(* Netzzustand Kaltwasser *)
IF Aktor_Netze_Anford.Kaltwasser.Aktiv THEN
	Zustand_Netz_KW.Temp_Max					:= MAX(Zustand_Netz_KW.Temp_Max, Aktor_Netze_Anford.Kaltwasser.Temp_Oben);
	Zustand_Netz_KW.Temp_Min					:= MIN(Zustand_Netz_KW.Temp_Min, Aktor_Netze_Anford.Kaltwasser.Temp_Unten);
	Zustand_Netz_KW.Regelung_Sollw_Oben_Max	:= MIN( Zustand_Netz_KW.Regelung_Sollw_Oben_Max, Aktor_Netze_Anford.Kaltwasser.Temp_Oben_Max);
	Zustand_Netz_KW.Regelung_Sollw_Oben_Min		:= MAX( Zustand_Netz_KW.Regelung_Sollw_Oben_Min, Aktor_Netze_Anford.Kaltwasser.Temp_Oben_Min);
	Zustand_Netz_KW.Regelung_Sollw_Unten_Max	:= MIN( Zustand_Netz_KW.Regelung_Sollw_Unten_Max, Aktor_Netze_Anford.Kaltwasser.Temp_Unten_Max);
	Zustand_Netz_KW.Regelung_Sollw_Unten_Min	:= MAX( Zustand_Netz_KW.Regelung_Sollw_Unten_Min, Aktor_Netze_Anford.Kaltwasser.Temp_Unten_Max);
END_IF
(* Netzzustand Warmwasser *)
IF Aktor_Netze_Anford.Warmwasser.Aktiv THEN
	Zustand_Netz_WW.Temp_Max					:= MAX(Zustand_Netz_WW.Temp_Max, Aktor_Netze_Anford.Kaltwasser.Temp_Oben);
	Zustand_Netz_WW.Temp_Min					:= MIN(Zustand_Netz_WW.Temp_Min, Aktor_Netze_Anford.Kaltwasser.Temp_Unten);
	Zustand_Netz_WW.Regelung_Sollw_Oben_Max	:= MIN( Zustand_Netz_WW.Regelung_Sollw_Oben_Max, Aktor_Netze_Anford.Kaltwasser.Temp_Oben_Max);
	Zustand_Netz_WW.Regelung_Sollw_Oben_Min	:= MAX( Zustand_Netz_WW.Regelung_Sollw_Oben_Min, Aktor_Netze_Anford.Kaltwasser.Temp_Oben_Min);
	Zustand_Netz_WW.Regelung_Sollw_Unten_Max	:= MIN( Zustand_Netz_WW.Regelung_Sollw_Unten_Max, Aktor_Netze_Anford.Kaltwasser.Temp_Unten_Max);
	Zustand_Netz_WW.Regelung_Sollw_Unten_Min	:= MAX( Zustand_Netz_WW.Regelung_Sollw_Unten_Min, Aktor_Netze_Anford.Kaltwasser.Temp_Unten_Max);
END_IF
(* Netzzustand Heisswasser *)
IF Aktor_Netze_Anford.Heisswasser.Aktiv THEN
	Zustand_Netz_HW.Temp_Max					:= MAX(Zustand_Netz_HW.Temp_Max, Aktor_Netze_Anford.Kaltwasser.Temp_Oben);
	Zustand_Netz_HW.Temp_Min					:= MIN(Zustand_Netz_HW.Temp_Min, Aktor_Netze_Anford.Kaltwasser.Temp_Unten);
	Zustand_Netz_HW.Regelung_Sollw_Oben_Max	:= MIN( Zustand_Netz_HW.Regelung_Sollw_Oben_Max, Aktor_Netze_Anford.Kaltwasser.Temp_Oben_Max);
	Zustand_Netz_HW.Regelung_Sollw_Oben_Min	:= MAX( Zustand_Netz_HW.Regelung_Sollw_Oben_Min, Aktor_Netze_Anford.Kaltwasser.Temp_Oben_Min);
	Zustand_Netz_HW.Regelung_Sollw_Unten_Max	:= MIN( Zustand_Netz_HW.Regelung_Sollw_Unten_Max, Aktor_Netze_Anford.Kaltwasser.Temp_Unten_Max);
	Zustand_Netz_HW.Regelung_Sollw_Unten_Min	:= MAX( Zustand_Netz_HW.Regelung_Sollw_Unten_Min, Aktor_Netze_Anford.Kaltwasser.Temp_Unten_Max);
END_IF;

Hysterese_Parameter.tTaskCycleTime	:= GA_global.Zeit_TaskCycle;
Hysterese_Parameter.tCtrlCycleTime		:= DINT_TO_TIME(Parameter.Kennlinie_Tctr);
Hysterese_Parameter.fHysteresisRange	:= 1;	(* 1 K *)

(* Initialisieren *)
Zustand.EIN_Anford		:= FALSE;
Zustand.EIN_Prioritaet		:= 0;
Zustand.AUS_Anford		:= FALSE;
Zustand.AUS_Prioritaet		:= 0;

(* Netzregelung Kaltwasser *)
IF( Parameter.Regelung_Netz_KW.Heizung AND Stellwert_Netz_KW.Leistung > 0 ) THEN
	Hysterese_Parameter.fHysteresisRange	:= Parameter.Regelung_Netz_KW.Hysterese_Heizung;
	Hysterese_KW_Heizung(
		fSetpointValue	:= Parameter.Regelung_Netz_KW.Grenzwert_Heizung,
		fActualValue		:= Stellwert_Netz_KW.Leistung,
		bSync			:= FALSE,
		eMode			:= eCTRL_MODE_ACTIVE,
		stParams		:= Hysterese_Parameter
	);
	IF( Hysterese_KW_Heizung.bOut ) THEN
		IF( Parameter.Regelung_Netz_KW.Invertiert_Heizung AND Parameter.Regelung_Netz_KW.Prioritaet_Heizung >= Zustand.AUS_Prioritaet) THEN
			Zustand.AUS_Anford		:= TRUE;
			Zustand.AUS_Prioritaet		:= Parameter.Regelung_Netz_KW.Prioritaet_Heizung;
		ELSIF( NOT Parameter.Regelung_Netz_KW.Invertiert_Heizung AND Parameter.Regelung_Netz_KW.Prioritaet_Heizung >= Zustand.EIN_Prioritaet) THEN
			Zustand.EIN_Anford		:= TRUE;
			Zustand.EIN_Prioritaet		:= Parameter.Regelung_Netz_KW.Prioritaet_Heizung;
		END_IF;
	END_IF;
ELSIF( Parameter.Regelung_Netz_KW.Heizung AND Stellwert_Netz_KW.Leistung < 0 ) THEN
	Hysterese_Parameter.fHysteresisRange	:= Parameter.Regelung_Netz_KW.Hysterese_Kuehlung;
	Hysterese_KW_Kuehlung(
		fSetpointValue	:= (-1) * Parameter.Regelung_Netz_KW.Grenzwert_Kuehlung,
		fActualValue		:= (-1) * Stellwert_Netz_KW.Leistung,
		bSync			:= FALSE,
		eMode			:= eCTRL_MODE_ACTIVE,
		stParams		:= Hysterese_Parameter
	);
	IF( Hysterese_KW_Kuehlung.bOut ) THEN
		IF( Parameter.Regelung_Netz_KW.Invertiert_Kuehlung AND Parameter.Regelung_Netz_KW.Prioritaet_Kuehlung >= Zustand.AUS_Prioritaet) THEN
			Zustand.AUS_Anford		:= TRUE;
			Zustand.AUS_Prioritaet		:= Parameter.Regelung_Netz_KW.Prioritaet_Kuehlung;
		ELSIF( NOT Parameter.Regelung_Netz_KW.Invertiert_Kuehlung AND Parameter.Regelung_Netz_KW.Prioritaet_Kuehlung >= Zustand.EIN_Prioritaet) THEN
			Zustand.EIN_Anford		:= TRUE;
			Zustand.EIN_Prioritaet		:= Parameter.Regelung_Netz_KW.Prioritaet_Kuehlung;
		END_IF;
	END_IF;
END_IF;

(* Netzregelung Warmwasser *)
IF( Parameter.Regelung_Netz_WW.Heizung AND Stellwert_Netz_WW.Leistung > 0 ) THEN
	Hysterese_Parameter.fHysteresisRange	:= Parameter.Regelung_Netz_WW.Hysterese_Heizung;
	Hysterese_WW_Heizung(
		fSetpointValue	:= Parameter.Regelung_Netz_WW.Grenzwert_Heizung,
		fActualValue		:= Stellwert_Netz_WW.Leistung,
		bSync			:= FALSE,
		eMode			:= eCTRL_MODE_ACTIVE,
		stParams		:= Hysterese_Parameter
	);
	IF( Hysterese_WW_Heizung.bOut ) THEN
		IF( Parameter.Regelung_Netz_WW.Invertiert_Heizung AND Parameter.Regelung_Netz_WW.Prioritaet_Heizung >= Zustand.AUS_Prioritaet) THEN
			Zustand.AUS_Anford		:= TRUE;
			Zustand.AUS_Prioritaet		:= Parameter.Regelung_Netz_WW.Prioritaet_Heizung;
		ELSIF( NOT Parameter.Regelung_Netz_WW.Invertiert_Heizung AND Parameter.Regelung_Netz_WW.Prioritaet_Heizung >= Zustand.EIN_Prioritaet) THEN
			Zustand.EIN_Anford		:= TRUE;
			Zustand.EIN_Prioritaet		:= Parameter.Regelung_Netz_WW.Prioritaet_Heizung;
		END_IF;
	END_IF;
ELSIF( Parameter.Regelung_Netz_WW.Heizung AND Stellwert_Netz_WW.Leistung < 0 ) THEN
	Hysterese_Parameter.fHysteresisRange	:= Parameter.Regelung_Netz_WW.Hysterese_Kuehlung;
	Hysterese_WW_Kuehlung(
		fSetpointValue	:= (-1) * Parameter.Regelung_Netz_WW.Grenzwert_Kuehlung,
		fActualValue		:= (-1) * Stellwert_Netz_WW.Leistung,
		bSync			:= FALSE,
		eMode			:= eCTRL_MODE_ACTIVE,
		stParams		:= Hysterese_Parameter
	);
	IF( Hysterese_WW_Kuehlung.bOut ) THEN
		IF( Parameter.Regelung_Netz_WW.Invertiert_Kuehlung AND Parameter.Regelung_Netz_WW.Prioritaet_Kuehlung >= Zustand.AUS_Prioritaet) THEN
			Zustand.AUS_Anford		:= TRUE;
			Zustand.AUS_Prioritaet		:= Parameter.Regelung_Netz_WW.Prioritaet_Kuehlung;
		ELSIF( NOT Parameter.Regelung_Netz_WW.Invertiert_Kuehlung AND Parameter.Regelung_Netz_WW.Prioritaet_Kuehlung >= Zustand.EIN_Prioritaet) THEN
			Zustand.EIN_Anford		:= TRUE;
			Zustand.EIN_Prioritaet		:= Parameter.Regelung_Netz_WW.Prioritaet_Kuehlung;
		END_IF;
	END_IF;
END_IF;

(* Netzregelung Heisswasser *)
IF( Parameter.Regelung_Netz_HW.Heizung AND Stellwert_Netz_HW.Leistung > 0 ) THEN
	Hysterese_Parameter.fHysteresisRange	:= Parameter.Regelung_Netz_HW.Hysterese_Heizung;
	Hysterese_HW_Heizung(
		fSetpointValue	:= Parameter.Regelung_Netz_HW.Grenzwert_Heizung,
		fActualValue		:= Stellwert_Netz_HW.Leistung,
		bSync			:= FALSE,
		eMode			:= eCTRL_MODE_ACTIVE,
		stParams		:= Hysterese_Parameter
	);
	IF( Hysterese_HW_Heizung.bOut ) THEN
		IF( Parameter.Regelung_Netz_HW.Invertiert_Heizung AND Parameter.Regelung_Netz_HW.Prioritaet_Heizung >= Zustand.AUS_Prioritaet) THEN
			Zustand.AUS_Anford		:= TRUE;
			Zustand.AUS_Prioritaet		:= Parameter.Regelung_Netz_HW.Prioritaet_Heizung;
		ELSIF( NOT Parameter.Regelung_Netz_HW.Invertiert_Heizung AND Parameter.Regelung_Netz_HW.Prioritaet_Heizung >= Zustand.EIN_Prioritaet) THEN
			Zustand.EIN_Anford		:= TRUE;
			Zustand.EIN_Prioritaet		:= Parameter.Regelung_Netz_HW.Prioritaet_Heizung;
		END_IF;
	END_IF;
ELSIF( Parameter.Regelung_Netz_HW.Heizung AND Stellwert_Netz_HW.Leistung < 0 ) THEN
	Hysterese_Parameter.fHysteresisRange	:= Parameter.Regelung_Netz_HW.Hysterese_Kuehlung;
	Hysterese_HW_Kuehlung(
		fSetpointValue	:= (-1) * Parameter.Regelung_Netz_HW.Grenzwert_Kuehlung,
		fActualValue		:= (-1) * Stellwert_Netz_HW.Leistung,
		bSync			:= FALSE,
		eMode			:= eCTRL_MODE_ACTIVE,
		stParams		:= Hysterese_Parameter
	);
	IF( Hysterese_HW_Kuehlung.bOut ) THEN
		IF( Parameter.Regelung_Netz_HW.Invertiert_Kuehlung AND Parameter.Regelung_Netz_HW.Prioritaet_Kuehlung >= Zustand.AUS_Prioritaet) THEN
			Zustand.AUS_Anford		:= TRUE;
			Zustand.AUS_Prioritaet		:= Parameter.Regelung_Netz_HW.Prioritaet_Kuehlung;
		ELSIF( NOT Parameter.Regelung_Netz_HW.Invertiert_Kuehlung AND Parameter.Regelung_Netz_HW.Prioritaet_Kuehlung >= Zustand.EIN_Prioritaet) THEN
			Zustand.EIN_Anford		:= TRUE;
			Zustand.EIN_Prioritaet		:= Parameter.Regelung_Netz_HW.Prioritaet_Kuehlung;
		END_IF;
	END_IF;
END_IF;



(* Stellwert bestimmen *)
Stellwert.Betrieb	:= Zustand.EIN_Anford AND NOT (Zustand.AUS_Anford AND (Zustand.AUS_Prioritaet > Zustand.EIN_Prioritaet));

END_FUNCTION_BLOCK

// ---- POUs/Management/FB_MGMT_Logik.TcPOU


FUNCTION_BLOCK FB_MGMT_Logik
VAR_IN_OUT
	Steuerung	: ST_FB_MGMT_Steuerung;
	Zustand		: ST_FB_MGMT_Zustand;
END_VAR
VAR_INPUT
	Parameter	: ST_FB_MGMT_Parameter;
END_VAR
VAR_OUTPUT
END_VAR
VAR
END_VAR

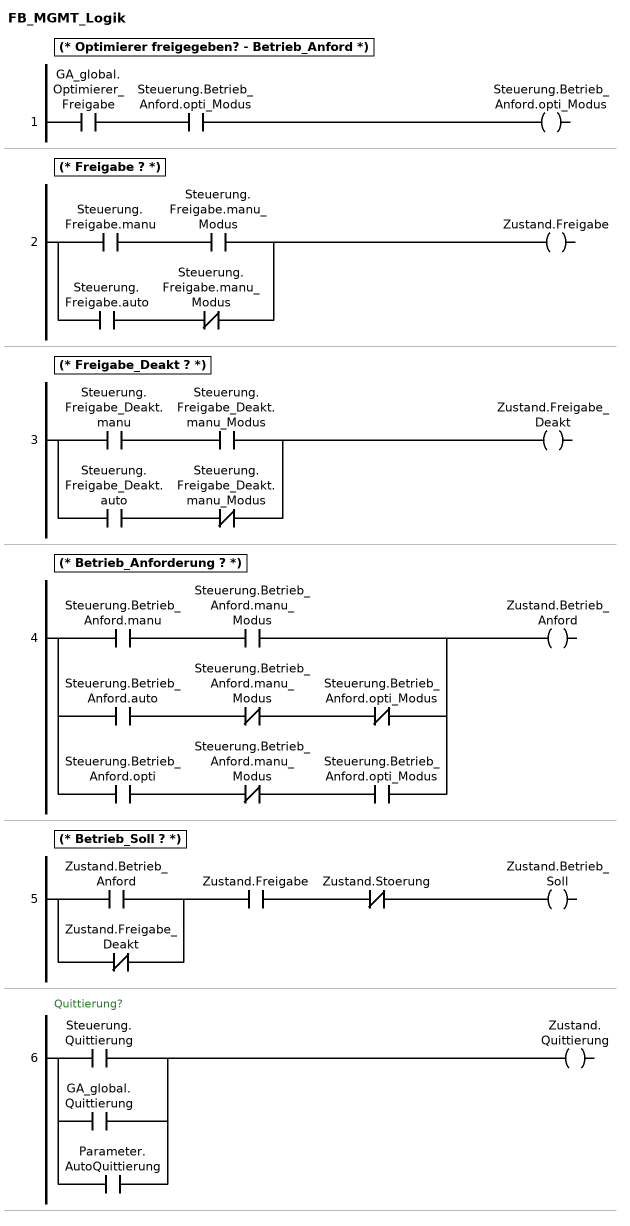
// NETWORK 1
// label: (* Optimierer freigegeben? - Betrieb_Anford *)
Steuerung.Betrieb_Anford.opti_Modus := GA_global.Optimierer_Freigabe AND Steuerung.Betrieb_Anford.opti_Modus;

// NETWORK 2
// label: (* Freigabe ? *)
Zustand.Freigabe := Steuerung.Freigabe.manu AND Steuerung.Freigabe.manu_Modus OR Steuerung.Freigabe.auto AND NOT Steuerung.Freigabe.manu_Modus;

// NETWORK 3
// label: (* Freigabe_Deakt ? *)
Zustand.Freigabe_Deakt := Steuerung.Freigabe_Deakt.manu AND Steuerung.Freigabe_Deakt.manu_Modus OR Steuerung.Freigabe_Deakt.auto AND NOT Steuerung.Freigabe_Deakt.manu_Modus;

// NETWORK 4
// label: (* Betrieb_Anforderung ? *)
Zustand.Betrieb_Anford := Steuerung.Betrieb_Anford.manu AND Steuerung.Betrieb_Anford.manu_Modus OR Steuerung.Betrieb_Anford.auto AND NOT Steuerung.Betrieb_Anford.manu_Modus AND NOT Steuerung.Betrieb_Anford.opti_Modus OR Steuerung.Betrieb_Anford.opti AND NOT Steuerung.Betrieb_Anford.manu_Modus AND Steuerung.Betrieb_Anford.opti_Modus;

// NETWORK 5
// label: (* Betrieb_Soll ? *)
Zustand.Betrieb_Soll := (Zustand.Betrieb_Anford OR NOT Zustand.Freigabe_Deakt) AND Zustand.Freigabe AND NOT Zustand.Stoerung;

// NETWORK 6
// Quittierung?
Zustand.Quittierung := Steuerung.Quittierung OR GA_global.Quittierung OR Parameter.AutoQuittierung;

END_FUNCTION_BLOCK

// ---- POUs/Management/FB_MGMT_Ablaufsteuerung.TcPOU
FUNCTION_BLOCK FB_MGMT_Ablaufsteuerung
VAR_IN_OUT
	Zustand				: ST_FB_MGMT_Zustand;
	Stellwert			: ST_FB_MGMT_Stellwert;
	Steuerung			: ST_FB_MGMT_Steuerung;
END_VAR
VAR_INPUT
END_VAR
VAR_OUTPUT
END_VAR
VAR
END_VAR

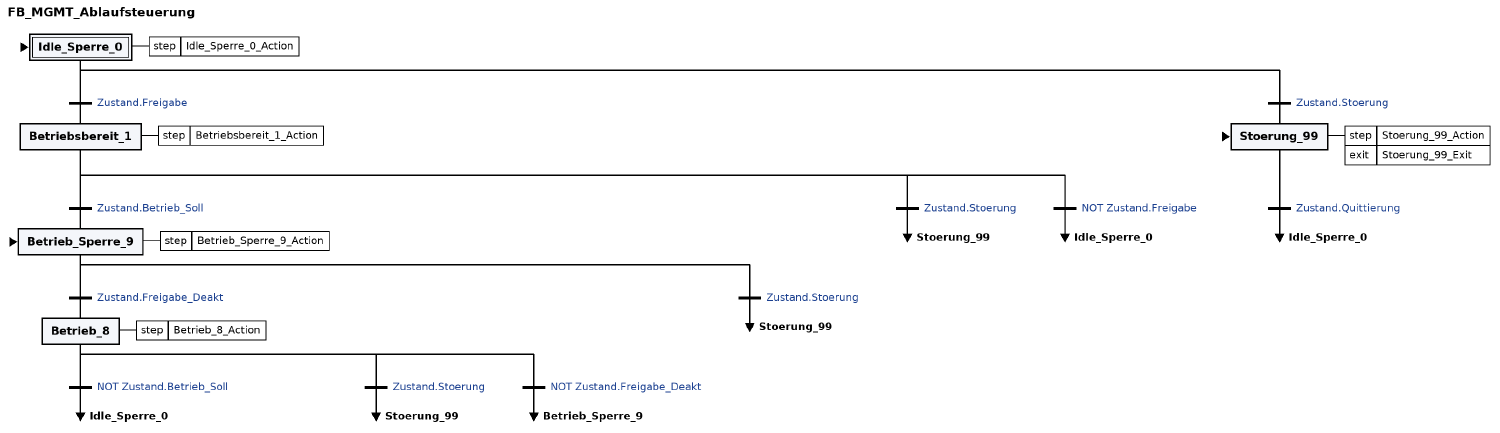
INITIAL_STEP Idle_Sperre_0:
    Idle_Sperre_0_Action(N);  // step action
END_STEP
TRANSITION FROM Idle_Sperre_0 TO Betriebsbereit_1
    := Zustand.Freigabe;
END_TRANSITION
TRANSITION FROM Idle_Sperre_0 TO Stoerung_99
    := Zustand.Stoerung;
END_TRANSITION
STEP Stoerung_99:
    Stoerung_99_Action(N);  // step action
    Stoerung_99_Exit(P0);  // exit action
END_STEP
TRANSITION FROM Stoerung_99 TO Idle_Sperre_0
    := Zustand.Quittierung;
END_TRANSITION
STEP Betriebsbereit_1:
    Betriebsbereit_1_Action(N);  // step action
END_STEP
TRANSITION FROM Betriebsbereit_1 TO Betrieb_Sperre_9
    := Zustand.Betrieb_Soll;
END_TRANSITION
TRANSITION FROM Betriebsbereit_1 TO Stoerung_99
    := Zustand.Stoerung;
END_TRANSITION
TRANSITION FROM Betriebsbereit_1 TO Idle_Sperre_0
    := NOT Zustand.Freigabe;
END_TRANSITION
STEP Betrieb_Sperre_9:
    Betrieb_Sperre_9_Action(N);  // step action
END_STEP
TRANSITION FROM Betrieb_Sperre_9 TO Betrieb_8
    := Zustand.Freigabe_Deakt;
END_TRANSITION
TRANSITION FROM Betrieb_Sperre_9 TO Stoerung_99
    := Zustand.Stoerung;
END_TRANSITION
STEP Betrieb_8:
    Betrieb_8_Action(N);  // step action
END_STEP
TRANSITION FROM Betrieb_8 TO Idle_Sperre_0
    := NOT Zustand.Betrieb_Soll;
END_TRANSITION
TRANSITION FROM Betrieb_8 TO Stoerung_99
    := Zustand.Stoerung;
END_TRANSITION
TRANSITION FROM Betrieb_8 TO Betrieb_Sperre_9
    := NOT Zustand.Freigabe_Deakt;
END_TRANSITION

ACTION Betrieb_8_Action:
(* Stellwert setzen *)
Stellwert.Betrieb				:= TRUE;
Zustand.Betrieb				:= TRUE;

(* Zustand setzen *)
Zustand.Status				:= E_MGMT_Zustand_Status_Betrieb;
END_ACTION

ACTION Betrieb_Sperre_9_Action:
(* Stellwert setzen *)
Stellwert.Betrieb				:= TRUE;
Zustand.Betrieb				:= TRUE;

(* Zustand setzen *)
Zustand.Status				:= E_MGMT_Zustand_Status_Betrieb_Sperre;
END_ACTION

ACTION Betriebsbereit_1_Action:
(* Stellwert setzen *)
Stellwert.Betrieb		:= FALSE;
Zustand.Betrieb		:= FALSE;

(* Zustand setzen *)
Zustand.Status			:= E_MGMT_Zustand_Status_Betriebsbereit;
END_ACTION

ACTION Idle_Sperre_0_Action:
(* Stellwert setzen *)
Stellwert.Betrieb		:= FALSE;
Zustand.Betrieb			:= FALSE;

(* Zustand setzen *)
Zustand.Status				:= E_MGMT_Zustand_Status_Idle_Sperre;

(* Quittierungszustand auf False setzen, damit das System bei einer erneuten Störung nicht direkt wieder angeschaltet wird *)
Steuerung.Quittierung	:= FALSE;
END_ACTION

ACTION Stoerung_99_Action:
(* Stellwert setzen *)
Stellwert.Betrieb			:= FALSE;
Zustand.Betrieb			:= FALSE;

(* Zustand setzen *)
Zustand.Stoerung			:= TRUE;
Zustand.Status			:= E_MGMT_Zustand_Status_Stoerung;
END_ACTION

ACTION Stoerung_99_Exit:
Zustand.Stoerung	:= FALSE;
END_ACTION

END_FUNCTION_BLOCK

// ---- POUs/Management/FB_MGMT_Sollwertscheck.TcPOU
FUNCTION_BLOCK FB_MGMT_Sollwertscheck
VAR_IN_OUT
	Zustand		: ST_FB_MGMT_Zustand;
END_VAR
VAR_INPUT
	Steuerung	: ST_FB_MGMT_Steuerung;
	Parameter	: ST_FB_MGMT_Parameter;
END_VAR
VAR

END_VAR

(* Priorisierung Regelung_Modus *)
IF(Steuerung.Regelung_Modus.manu_Modus) THEN
	Zustand.Regelung_Modus := Steuerung.Regelung_Modus.manu;
ELSIF(Steuerung.Regelung_Modus.opti_Modus) THEN
	Zustand.Regelung_Modus := Steuerung.Regelung_Modus.opti;
ELSE
	Zustand.Regelung_Modus := Steuerung.Regelung_Modus.auto;
END_IF;
(* Priorisierung Regelung_Sollwert *)
IF(Steuerung.Regelung_Sollw.manu_Modus) THEN
	Zustand.Regelung_Sollw_Anford := Steuerung.Regelung_Sollw.manu;
ELSIF(Steuerung.Regelung_Sollw.opti_Modus) THEN
	Zustand.Regelung_Sollw_Anford := Steuerung.Regelung_Sollw.opti;
ELSE
	Zustand.Regelung_Sollw_Anford := Steuerung.Regelung_Sollw.auto;
END_IF;

(*Berechnung Sollwert mithilfe von Netze*)

(*Heizen*)

Zustand.Regelung_Sollw_BHKW_WBZ := Zustand.Heisswasser_3xx_Zustand_Regelung_Sollw;
Zustand.Regelung_Sollw_BHKW_MBZ := Zustand.Heisswasser_3xx_Zustand_Regelung_Sollw - 2;
Zustand.Regelung_Sollw_BWT:= Zustand.Heisswasser_3xx_Zustand_Regelung_Sollw - 4;

(*Warmnetz*)
Zustand.Regelung_Sollw_PTW1:= Zustand.Warmwasser_2xx_Zustand_Regelung_Sollw;
Zustand.Regelung_Sollw_WP_gruennetz :=  Zustand.Warmwasser_2xx_Zustand_Regelung_Sollw - 3;
Zustand.Regelung_Sollw_gruennetz_Kuehlung:=Zustand.Warmwasser_2xx_Zustand_Regelung_Sollw_Max;


(*Kühlen*)
Zustand.Regelung_Sollw_blaunetz_Kuehlung:= Zustand.Kaltwasser_1xx_Zustand_Regelung_Sollw;
Zustand.Regelung_Sollw_Kuehlung_KKKW := MIN(Zustand.Kaltwasser_1xx_Zustand_Regelung_Sollw + 3, Zustand.Temp_KRITIKAL_OBEN_TEMP_Kaltnetz)  ;
Zustand.Regelung_Sollw_WP_945 := MAX(Zustand.Kaltwasser_1xx_Zustand_Regelung_Sollw, Zustand.Temp_KRITIKAL_UNTEN_TEMP_Kaltnetz );

END_FUNCTION_BLOCK

// ---- POUs/Management/FB_MGMT_Regelung.TcPOU
FUNCTION_BLOCK FB_MGMT_Regelung
VAR_IN_OUT
	Stellwert	: ST_FB_MGMT_Stellwert;
	Zustand		: ST_FB_MGMT_Zustand;
END_VAR
VAR_INPUT
	Steuerung	: ST_FB_MGMT_Steuerung;
	Parameter	: ST_FB_MGMT_Parameter;
END_VAR
VAR_OUTPUT
END_VAR
VAR
(*Hysterese Heizung*)
	Hysterese_BHKW_MBZ 					: FB_CTRL_2POINT; (*BHKW mit mehrerer Betriebzeit*)
	Hysterese_Parameter_BHKW_MBZ		: ST_CTRL_2POINT_PARAMS; (*BHKW mit mehrerer Betriebzeit*)
	Hysterese_BHKW_WBZ 					: FB_CTRL_2POINT; (*BHKW mit wenigerer Betriebzeit*)
	Hysterese_Parameter_BHKW_WBZ 		: ST_CTRL_2POINT_PARAMS; (*BHKW mit wenigerer Betriebzeit*)
	Hysterese_PWT_915 					: FB_CTRL_2POINT;
	Hysterese_Parameter_PWT_915 		: ST_CTRL_2POINT_PARAMS;
	Hysterese_BWT 						: FB_CTRL_2POINT;
	Hysterese_Parameter_BWT		 		: ST_CTRL_2POINT_PARAMS;
	Hysterese_WP_gruennetz				: FB_CTRL_2POINT;
	Hysterese_Parameter_WP_gruennetz	: ST_CTRL_2POINT_PARAMS;

(*Hysterese Kuehlung*)
	Hysterese_Kuehlung_KKKW                 : FB_CTRL_2POINT;
    Hysterese_Parameter_Kuehlung_KKKW       : ST_CTRL_2POINT_PARAMS;
	Hysterese_WP_945						: FB_CTRL_2POINT;
	Hysterese_Parameter_WP_945				: ST_CTRL_2POINT_PARAMS;

	WaermePumpe_Anforderung_gruennetz: BOOL;
	WaermePumpe_Anforderung_blaunetz: BOOL;

	Hysterese_BHKW_921: BOOL;
	t: REAL;
	Wechsel_Erlaubnis: BOOL; (*wenn Wechsel_Erlaubnis==true ist, dann darf Wechsel zwischen Hysterese erfolgen. Wechsel_Erlaubnis wird erst nach 24 Stunden nach dem letzten Wechsel True*)
	tstunde: REAL; (*Wenn die Hysterese für BHKW gewechselt werden*)
	ttag: REAL; (*Wenn die Hysterese für BHKW gewechselt werden*)
    aktuell_Modus: INT; (*Wenn diese Variable 1 ist, dann Output.BHKW2=MBZ und wenn 2 ist, dann Output.BHKW1=WBZ*)

    Kuehlung_Erlaubnis_KKKW    : BOOL; (*Wenn die Isttemperatur vom blauen Netz ist mehr als 3 Grad mehr als Solltemperatur, dann Chiller wird abgeschaltet. *)
END_VAR

(*Hysterese_Regelung für BHKW_MBZ(BHKW mit mehrerer Betriebzeit), Hysterese von Zustand.Regelung_Sollw_BHKW_MBZ-Range/2 bis Zustand.Regelung_Sollw_BHKW_MBZ+Range/2 °C*)

Hysterese_Parameter_BHKW_MBZ.fHysteresisRange := Parameter.Hysterese_BHKW_Range;
Hysterese_Parameter_BHKW_MBZ.tTaskCycleTime	:= GA_global.Zeit_TaskCycle; (* Zykluszeit FB = globaler Zykluszeit*)
Hysterese_Parameter_BHKW_MBZ.tCtrlCycleTime := GA_global.Zeit_TaskCycle;

Hysterese_BHKW_MBZ(
	fSetpointValue  := Zustand.Regelung_Sollw_BHKW_MBZ,
	fActualValue    := Zustand.Temp_Hysterese_BHKW_A,
	eMode			:= eCTRL_MODE_ACTIVE,
	stParams		:= Hysterese_Parameter_BHKW_MBZ
);

(*Beim Aufheizen wird auf untere Temperatur geregelt, beim Abkühlen wird auf obere Temperatur geregelt.*)

IF (Hysterese_BHKW_MBZ.bOut) THEN
Zustand.Temp_Hysterese_BHKW_A := Zustand.Temp_Unten_Heissnetz;
ELSE
Zustand.Temp_Hysterese_BHKW_A := Zustand.Temp_Oben_Heissnetz;
END_IF

(*Hysterese_Regelung für BHKW_WBZ(BHKW mit wenigerer Betriebzeit), Hysterese von Zustand.Regelung_Sollw_BHKW_WBZ-Range/2 bis Zustand.Regelung_Sollw_BHKW_WBZ+Range/2 °C*)

Hysterese_Parameter_BHKW_WBZ.fHysteresisRange := Parameter.Hysterese_BHKW_Range;
Hysterese_Parameter_BHKW_WBZ.tTaskCycleTime	:= GA_global.Zeit_TaskCycle; (* Zykluszeit FB = globaler Zykluszeit*)
Hysterese_Parameter_BHKW_WBZ.tCtrlCycleTime := GA_global.Zeit_TaskCycle;

Hysterese_BHKW_WBZ(
	fSetpointValue  := Zustand.Regelung_Sollw_BHKW_WBZ,
	fActualValue    := Zustand.Temp_Hysterese_BHKW_B,
	eMode			:= eCTRL_MODE_ACTIVE,
	stParams		:= Hysterese_Parameter_BHKW_WBZ
);

(*Beim Aufheizen wird auf untere Temperatur geregelt, beim Abkühlen wird auf obere Temperatur geregelt.*)

IF (Hysterese_BHKW_WBZ.bOut) THEN
Zustand.Temp_Hysterese_BHKW_B := Zustand.Temp_Unten_Heissnetz;
ELSE
Zustand.Temp_Hysterese_BHKW_B := Zustand.Temp_Oben_Heissnetz;
END_IF


(*BHKW mit wenigerer Betriebzeit übernimmt die höhere Hysterese*)

IF	(Wandler.System_Blockheizkraftwerk_922.BHKW_922.Zustand.Zeit_Betrieb>Wandler.System_Blockheizkraftwerk_921.BHKW_921.Zustand.Zeit_Betrieb) AND (Wechsel_Erlaubnis) THEN

Wechsel_Erlaubnis:=FALSE;
ttag:=GA_global.Systemzeit_Tag;
tstunde:=GA_global.Systemzeit_Stunde;
aktuell_Modus:=1;

ELSIF (Wandler.System_Blockheizkraftwerk_922.BHKW_922.Zustand.Zeit_Betrieb<Wandler.System_Blockheizkraftwerk_921.BHKW_921.Zustand.Zeit_Betrieb) AND (Wechsel_Erlaubnis) THEN

Wechsel_Erlaubnis:=FALSE;
ttag:=GA_global.Systemzeit_Tag;
tstunde:=GA_global.Systemzeit_Stunde;
aktuell_Modus:=2;

END_IF

CASE aktuell_Modus OF
1:
Stellwert.BHKW1_Anforderung := Hysterese_BHKW_WBZ.bOut;
Stellwert.BHKW2_Anforderung := Hysterese_BHKW_MBZ.bOut;

2:
Stellwert.BHKW1_Anforderung := Hysterese_BHKW_MBZ.bOut;
Stellwert.BHKW2_Anforderung := Hysterese_BHKW_WBZ.bOut;
END_CASE;

(*Wenn ein BHKW in Störung ist, dann übernimmt die andere seine Hysterese*)
IF (Zustand.BHKW921_Stoerung) AND (Stellwert.BHKW1_Anforderung) THEN
Stellwert.BHKW2_Anforderung := Stellwert.BHKW1_Anforderung;
ELSIF (Zustand.BHKW922_Stoerung) AND (Stellwert.BHKW2_Anforderung) THEN
Stellwert.BHKW1_Anforderung := Stellwert.BHKW2_Anforderung;
END_IF

(*Der Wechsel zwischen Hysterese darf nur einmal in 24 Stunden passieren.*)
t:= (GA_global.Systemzeit_Tag-ttag)*24 + GA_global.Systemzeit_Stunde-tstunde;

IF(t>24) THEN
Wechsel_Erlaubnis:=TRUE;
ELSE
Wechsel_Erlaubnis:= FALSE;
END_IF


(*Brennwerttherme an, Hysterese von Zustand.Regelung_Sollw_BWT-Range/2 bis Zustand.Regelung_Sollw_BWT+Range/2 °C*)
Hysterese_Parameter_BWT.fHysteresisRange := Parameter.Hysterese_BWT_Range;
Hysterese_Parameter_BWT.tTaskCycleTime	:= GA_global.Zeit_TaskCycle; (* Zykluszeit FB = globaler Zykluszeit*)
Hysterese_Parameter_BWT.tCtrlCycleTime := GA_global.Zeit_TaskCycle;

Hysterese_BWT(
	fSetpointValue  := Zustand.Regelung_Sollw_BWT,
	fActualValue    := Zustand.Temp_Hysterese_BWT,
	bSync			:= FALSE,
	eMode			:= eCTRL_MODE_ACTIVE,
	stParams		:= Hysterese_Parameter_BWT
);

Stellwert.BWT_Anforderung  := Hysterese_BWT.bOut;

(*Beim Aufheizen wird auf untere Temperatur geregelt, beim Abkühlen wird auf obere Temperatur geregelt.*)

IF (Hysterese_BWT.bOut) THEN
Zustand.Temp_Hysterese_BWT := Zustand.Temp_Unten_Heissnetz;
ELSE
Zustand.Temp_Hysterese_BWT := Zustand.Temp_Oben_Heissnetz;
END_IF


(*Wärmetauscher an, Hysterese von  Zustand.Regelung_Sollw_PTW1-Range/2 bis  Zustand.Regelung_Sollw_PTW1+Range/2 °C*)

Hysterese_Parameter_PWT_915.fHysteresisRange := Parameter.Hysterese_PTW1_Range;
Hysterese_Parameter_PWT_915.tTaskCycleTime	:= GA_global.Zeit_TaskCycle; (* Zykluszeit FB = globaler Zykluszeit*)
Hysterese_Parameter_PWT_915.tCtrlCycleTime := GA_global.Zeit_TaskCycle;

Hysterese_PWT_915(
	fSetpointValue  := Zustand.Regelung_Sollw_PTW1,
	fActualValue    := Zustand.Temp_Unten_Warmnetz,
	bSync			:= FALSE,
	eMode			:= eCTRL_MODE_ACTIVE,
	stParams		:= Hysterese_Parameter_PWT_915
);

Stellwert.PWT1_Anforderung  := Hysterese_PWT_915.bOut;

(*Wärmepumpe kannzum Kühlen des blauen Netzes oder zum Aufwärmen des gelben Netzes benutzt werden*)
(*Wärmepumpe an, Hysterese Regelung von Zustand.Regelung_Sollw_WP_gruennetz-Range/2 bis Zustand.Regelung_Sollw_WP_gruennetz+Range/2 °C*)



Hysterese_Parameter_WP_gruennetz.fHysteresisRange := Parameter.Hysterese_WP_gruennetz_Range;
Hysterese_Parameter_WP_gruennetz.tTaskCycleTime	:= GA_global.Zeit_TaskCycle; (* Zykluszeit FB = globaler Zykluszeit*)
Hysterese_Parameter_WP_gruennetz.tCtrlCycleTime := GA_global.Zeit_TaskCycle;

Hysterese_WP_gruennetz(
	fSetpointValue  := Zustand.Regelung_Sollw_WP_gruennetz,
	fActualValue    := Zustand.Temp_Unten_Warmnetz,
	bSync			:= FALSE,
	eMode			:= eCTRL_MODE_ACTIVE,
	stParams		:= Hysterese_Parameter_WP_gruennetz
);

(*Wenn die Temperatur des Balunetzes weniger als Kritikal_Unten_Temp ist, dann müssen Wärmepumpe ausgeschaltet werden*)
WaermePumpe_Anforderung_gruennetz  := Hysterese_WP_gruennetz.bOut AND (Zustand.Temp_Unten_Kaltnetz>Zustand.Temp_KRITIKAL_UNTEN_TEMP_Kaltnetz);


(*Hysterese_Regelung für Wärmepumpe blaunetz_Kuehlung*)
Hysterese_Parameter_WP_945.fHysteresisRange := Parameter.Hysterese_WP_Range;
Hysterese_Parameter_WP_945.tTaskCycleTime	:= GA_global.Zeit_TaskCycle;	(* Zykluszeit FB = globaler Zykluszeit*)
Hysterese_Parameter_WP_945.tCtrlCycleTime	:= GA_global.Zeit_TaskCycle;

Hysterese_WP_945(
	fSetpointValue 	:= Zustand.Regelung_Sollw_WP_945 - 1,
	fActualValue    := Zustand.Temp_Oben_Kaltnetz,
	bSync			:= FALSE,
	eMode			:= eCTRL_MODE_ACTIVE,
	stParams 		:= Hysterese_Parameter_WP_945
);

(*Wenn die Temperatur des Gruennetzes mehr als Kritikal_Oben_Temp ist, dann müssen Wärmepumpe ausgeschaltet werden*)
WaermePumpe_Anforderung_blaunetz := NOT Hysterese_WP_945.bOut AND NOT Hysterese_WP_945.bError AND (Zustand.Temp_Oben_Warmnetz<Zustand.Temp_KRITIKAL_OBEN_TEMP_Warmnetz) ;

Stellwert.Waermepumpe_945_Anforderung :=  WaermePumpe_Anforderung_gruennetz OR WaermePumpe_Anforderung_blaunetz;

(*Hysterese_Regelung für Kältekompressor Kaltwasser*)

Hysterese_Parameter_Kuehlung_KKKW.fHysteresisRange :=Parameter.Hysterese_KKKW_Kuehlung_Range;
Hysterese_Parameter_Kuehlung_KKKW.tTaskCycleTime	:= GA_global.Zeit_TaskCycle; (* Zykluszeit FB = globaler Zykluszeit*)
Hysterese_Parameter_Kuehlung_KKKW.tCtrlCycleTime := GA_global.Zeit_TaskCycle;

Hysterese_Kuehlung_KKKW(
	fSetpointValue  := Zustand.Regelung_Sollw_Kuehlung_KKKW,
	fActualValue    := Zustand.Temp_Oben_Kaltnetz,
	bSync			:= FALSE,
	eMode			:= eCTRL_MODE_ACTIVE,
	stParams		:= Hysterese_Parameter_Kuehlung_KKKW
);

(*Wenn die Kühlleistung vom Speicher nicht reicht, dann schaltet der Chiller an*)

IF (Zustand.Temp_Oben_Kaltnetz-Zustand.Regelung_Sollw_blaunetz_Kuehlung>3) THEN
Kuehlung_Erlaubnis_KKKW := TRUE;
ELSE
Kuehlung_Erlaubnis_KKKW := FALSE;
END_IF

Stellwert.Kuehlung_KKKW_Anforderung := NOT Hysterese_Kuehlung_KKKW.bOut AND NOT Hysterese_Kuehlung_KKKW.bError AND Kuehlung_Erlaubnis_KKKW ;


(*Entziehen der Freigabe, wenn Kritikal ObenTemperatur überschritten wird*)
(*
IF (Zustand.Temp_Oben_Heissnetz>Zustand.Temp_KRITIKAL_OBEN_TEMP_Heissnetz) THEN

Stellwert.BHKW1_Freigabe_Entziehung := TRUE;
Stellwert.BHKW2_Freigabe_Entziehung := TRUE;
Stellwert.BWT_Freigabe_Entziehung := TRUE;
GA_global.Optimierer_Freigabe := FALSE;
ELSE
Stellwert.BHKW1_Freigabe_Entziehung := FALSE;
Stellwert.BHKW2_Freigabe_Entziehung := FALSE;
Stellwert.BWT_Freigabe_Entziehung := FALSE;
(*GA_global.Optimierer_Freigabe := TRUE;*)
END_IF

IF (Zustand.Temp_Oben_Warmnetz>Zustand.Temp_KRITIKAL_OBEN_TEMP_Warmnetz) THEN

Stellwert.PWT1_Freigabe_Entziehung := TRUE;
Stellwert.WP_Freigabe_Entziehung := TRUE;
GA_global.Optimierer_Freigabe := FALSE;

ELSE
Stellwert.PWT1_Freigabe_Entziehung := FALSE;
Stellwert.WP_Freigabe_Entziehung := FALSE;

END_IF

IF Zustand.Temp_Unten_Kaltnetz<Zustand.Temp_KRITIKAL_UNTEN_TEMP_Kaltnetz THEN
GA_global.Optimierer_Freigabe := FALSE;
END_IF
*)

END_FUNCTION_BLOCK

// ---- POUs/Management/FB_Zuweisungen.TcPOU
FUNCTION_BLOCK FB_Zuweisungen
VAR_INPUT
END_VAR
VAR_IN_OUT
	Zustand		: ST_FB_MGMT_Zustand;
END_VAR
VAR_OUTPUT
END_VAR
VAR
END_VAR

Zustand.Temp_Speicher795:= Speicher.System_Betonspeicher_Kaltwasser_795.Betonspeicher_795.Zustand.Temp_oben;
Zustand.Temp_Oben_Heissnetz :=Netze.Heisswasser_3xx.Zustand.Temp_Oben;
Zustand.Temp_Unten_Heissnetz:= Netze.Heisswasser_3xx.Zustand.Temp_Unten;
Zustand.Temp_Oben_Warmnetz:= Netze.Warmwasser_2xx.Zustand.Temp_Oben;
Zustand.Temp_Unten_Warmnetz:=Netze.Warmwasser_2xx.Zustand.Temp_Unten;
Zustand.Temp_Oben_Kaltnetz:=Netze.Kaltwasser_1xx.Zustand.Temp_Oben;
Zustand.Temp_Unten_Kaltnetz:=Netze.Kaltwasser_1xx.Zustand.Temp_Unten;
Zustand.BHKW921_Stoerung:=Wandler.System_Blockheizkraftwerk_921.Zustand.Stoerung;
Zustand.BHKW922_Stoerung:=Wandler.System_Blockheizkraftwerk_922.Zustand.Stoerung;
Zustand.Temp_KRITIKAL_OBEN_TEMP_Heissnetz:=Netze.Heisswasser_3xx.Parameter.Regelung_Sollw_KRITIKAL_OBEN_TEMP;
Zustand.Temp_KRITIKAL_OBEN_TEMP_Warmnetz:= Netze.Warmwasser_2xx.Parameter.Regelung_Sollw_KRITIKAL_OBEN_TEMP;
Zustand.Temp_KRITIKAL_OBEN_TEMP_Kaltnetz:=Netze.Kaltwasser_1xx.Parameter.Regelung_Sollw_KRITIKAL_OBEN_TEMP;
Zustand.Temp_KRITIKAL_UNTEN_TEMP_Heissnetz:=Netze.Heisswasser_3xx.Parameter.Regelung_Sollw_KRITIKAL_UNTEN_TEMP;
Zustand.Temp_KRITIKAL_UNTEN_TEMP_Warmnetz:= Netze.Warmwasser_2xx.Parameter.Regelung_Sollw_KRITIKAL_UNTEN_TEMP;
Zustand.Temp_KRITIKAL_UNTEN_TEMP_Kaltnetz:=Netze.Kaltwasser_1xx.Parameter.Regelung_Sollw_KRITIKAL_UNTEN_TEMP;

Zustand.Heisswasser_3xx_Zustand_Regelung_Sollw:= Netze.Heisswasser_3xx.Zustand.Regelung_Sollw;
Zustand.Warmwasser_2xx_Zustand_Regelung_Sollw:=Netze.Warmwasser_2xx.Zustand.Regelung_Sollw;
Zustand.Warmwasser_2xx_Zustand_Regelung_Sollw_Max := Netze.Warmwasser_2xx.Zustand.Regelung_Sollw_Max;
Zustand.Kaltwasser_1xx_Zustand_Regelung_Sollw:=Netze.Kaltwasser_1xx.Zustand.Regelung_Sollw;

END_FUNCTION_BLOCK

// ---- POUs/FB_Initialisierungsroutine.TcPOU
FUNCTION_BLOCK FB_Initialisierungsroutine
VAR_OUTPUT
END_VAR
VAR

END_VAR

(*Management Parameter*)

Initialisierung.MGMT_Parameter.Temp_Max :=100; (*Grad Celsius*)
Initialisierung.MGMT_Parameter.Temp_Min :=0; (*Grad Celsius*)
Initialisierung.MGMT_Parameter.AutoQuittierung := 0;

(*Management Parameter- Heizen*)

Initialisierung.MGMT_Parameter.Hysterese_BHKW_Range := 3; (*Grad Celsius*) (*Range von die Hysterese für BHKW*)
Initialisierung.MGMT_Parameter.Hysterese_BWT_Range := 5; (*Grad Celsius*) (*Range von die Hysterese für BWT*)
Initialisierung.MGMT_Parameter.Hysterese_PTW1_Range := 3; (*Grad Celsius*) (*Range von die Hysterese für PWT*)


(*Management Parameter- Kühlen*)
Initialisierung.MGMT_Parameter.Hysterese_blaunetz_Kuehlung_Range := 2; (*Grad Celsius*) (*Range von Blaunetz_Hysterese *)
Initialisierung.MGMT_Parameter.Hysterese_KKKW_Kuehlung_Range := 2; (*Grad Celsius*) (*Range von Kältekompressor_Hysterese*)
Initialisierung.MGMT_Parameter.Hysterese_gruennetz_Kuehlung_Range := 2; (*Grad Celsius*) (*Range von Grünnetz_Hysterese*)
Initialisierung.MGMT_Parameter.Hysterese_WP_gruennetz_Range := 2; (*Grad Celsius*) (*Range von Wärmepumpe für gruenNetz *)
Initialisierung.MGMT_Parameter.Hysterese_WP_Range := 2; (*Grad Celsius*) (*Range von Hysterese_Regelung für Wärmepumpe blau_kuehlmodus_Kuehlung*)

(*Netze Parameter*)
Initialisierung.Netze_Parameter.Heisswasser.Regelung_Sollw_Max_Min := 50; (*Grad Celsius*)
Initialisierung.Netze_Parameter.Heisswasser.Regelung_Sollw_Min := 30; (*Grad Celsius*)
Initialisierung.Netze_Parameter.Heisswasser.Regelung_Sollw_KRITIKAL_OBEN_TEMP := 90; (*Grad Celsius*)
Initialisierung.Netze_Parameter.Heisswasser.Regelung_Sollw_KRITIKAL_UNTEN_TEMP := 20; (*Grad Celsius*)
Initialisierung.Netze_Parameter.Warmwasser.Regelung_Sollw_Max := 45; (*Grad Celsius*)
Initialisierung.Netze_Parameter.Warmwasser.Regelung_Sollw_Min := 25; (*Grad Celsius*)
Initialisierung.Netze_Parameter.Warmwasser.Regelung_Sollw_KRITIKAL_OBEN_TEMP := 65; (*Grad Celsius*)
Initialisierung.Netze_Parameter.Warmwasser.Regelung_Sollw_KRITIKAL_UNTEN_TEMP := 15; (*Grad Celsius*)
Initialisierung.Netze_Parameter.Kaltwasser.Regelung_Sollw_Max := 25; (*Grad Celsius*)
Initialisierung.Netze_Parameter.Kaltwasser.Regelung_Sollw_KRITIKAL_OBEN_TEMP := 28; (*Grad Celsius*)
Initialisierung.Netze_Parameter.Kaltwasser.Regelung_Sollw_KRITIKAL_UNTEN_TEMP := 6; (*Grad Celsius*)

Initialisierung.Netze_Parameter.Heisswasser.Temp_Max := 100; (*Grad Celsius*)
Initialisierung.Netze_Parameter.Heisswasser.Temp_Min := 0; (*Grad Celsius*)

Initialisierung.Netze_Parameter.Heisswasser.AutoQuittierung := 0;
Initialisierung.Netze_Parameter.Warmwasser.AutoQuittierung := 0;
Initialisierung.Netze_Parameter.Kaltwasser.AutoQuittierung := 0;

(*Parameter System Aussenfassadenaktivierung *)
	Initialisierung.System_AFA_Parameter.AutoQuittierung := 0;
	Initialisierung.System_AFA_Parameter.Freigabe_Berieselung := FALSE;
	Initialisierung.System_AFA_Parameter.Temp_Vorl_Max := 45; (*Grad Celsius*)
	Initialisierung.System_AFA_Parameter.Temp_Vorl_Min := 4; (*Grad Celsius*)
	Initialisierung.System_AFA_Parameter.Zeit_Nachl := 30; (*Millisekunden*)

	Initialisierung.Stellventil_605_Parameter.AutoQuittierung := 0;
	Initialisierung.Stellventil_605_Parameter.Zeit_Stellen0 := 10000; (*Millisekunden*)
	Initialisierung.Stellventil_605_Parameter.Zeit_Stellen1 := 10000; (*Millisekunden*)

	Initialisierung.Stellventil_235_Parameter.AutoQuittierung := 0;
	Initialisierung.Stellventil_235_Parameter.Zeit_Stellen0 := 10000; (*Millisekunden*)
	Initialisierung.Stellventil_235_Parameter.Zeit_Stellen1 := 10000; (*Millisekunden*)

	Initialisierung.Pumpe_600_Parameter.AutoQuittierung := 0;
	Initialisierung.Pumpe_600_Parameter.Regelung_PI_Kp := 0.265; (*Einheitslos*)
	Initialisierung.Pumpe_600_Parameter.Regelung_PI_Tctr := 5000; (*Millisekunden*)
	Initialisierung.Pumpe_600_Parameter.Regelung_PI_Tn := 15000; (*Millisekunden*)
	Initialisierung.Pumpe_600_Parameter.Stellwert_Leistung_Max := 100; (*Prozent*)
	Initialisierung.Pumpe_600_Parameter.Stellwert_Leistung_Min := 30; (*Prozent*)
	Initialisierung.Pumpe_600_Parameter.Zeit_Nachl := 2000; (*Millisekunden*)
	Initialisierung.Pumpe_600_Parameter.Zeit_Vorl := 2000; (*Millisekunden*)

	Initialisierung.Pumpe_235_Parameter.AutoQuittierung := 0;
	Initialisierung.Pumpe_235_Parameter.Regelung_PI_Kp := 0.265; (*Einheitslos*)
	Initialisierung.Pumpe_235_Parameter.Regelung_PI_Tctr := 5000; (*Millisekunden*)
	Initialisierung.Pumpe_235_Parameter.Regelung_PI_Tn := 15000; (*Millisekunden*)
	Initialisierung.Pumpe_235_Parameter.Stellwert_Leistung_Max := 100; (*Prozent*)
	Initialisierung.Pumpe_235_Parameter.Stellwert_Leistung_Min := 30; (*Prozent*)
	Initialisierung.Pumpe_235_Parameter.Zeit_Nachl := 2000; (*Millisekunden*)
	Initialisierung.Pumpe_235_Parameter.Zeit_Vorl := 2000; (*Millisekunden*)

	Initialisierung.Regelventil_600_Parameter.AutoQuittierung := 0;
	Initialisierung.Regelventil_600_Parameter.Regelung_PI_Kp := 0.5;
	Initialisierung.Regelventil_600_Parameter.Regelung_PI_Tctr := 5000; (*Millisekunden*)
	Initialisierung.Regelventil_600_Parameter.Regelung_PI_Tn := 15000; (*Millisekunden*)
	Initialisierung.Regelventil_600_Parameter.Regelung_Sollw_Max := 35; (*Grad Celsius*)
	Initialisierung.Regelventil_600_Parameter.Regelung_Sollw_Min := 5; (*Grad Celsius*)
	Initialisierung.Regelventil_600_Parameter.Regelung_Sollw_Rampe_Steig_neg := 0.0055;(*Einheit: K/s,  0,0055 K/s ~ 20 K/h*)
	Initialisierung.Regelventil_600_Parameter.Regelung_Sollw_Rampe_Steig_pos := 0.0055;(*Einheit: K/s,  0,0055 K/s ~ 20 K/h*)
	Initialisierung.Regelventil_600_Parameter.Stellwert_Stellung_Max := 100; (*Prozent*)
	Initialisierung.Regelventil_600_Parameter.Stellwert_Stellung_Min := 0; (*Prozent*)
	Initialisierung.Regelventil_600_Parameter.Zeit_Nachl := 15000; (*Millisekunden*)
	Initialisierung.Regelventil_600_Parameter.Zeit_Vorl := 15000; (*Millisekunden*)

	Initialisierung.Regelventil_640_Parameter.AutoQuittierung := 0;
	Initialisierung.Regelventil_640_Parameter.Regelung_PI_Kp := 0.265; (*Einheitslos*)
	Initialisierung.Regelventil_640_Parameter.Regelung_PI_Tctr := 5000; (*Millisekunden*)
	Initialisierung.Regelventil_640_Parameter.Regelung_PI_Tn := 15000; (*Millisekunden*)
	Initialisierung.Regelventil_640_Parameter.Regelung_Sollw_Max := 35; (*Grad Celsius*)
	Initialisierung.Regelventil_640_Parameter.Regelung_Sollw_Min := 5;(*Grad Celsius*)
	Initialisierung.Regelventil_640_Parameter.Regelung_Sollw_Rampe_Steig_neg := 0.0055;(*Einheit: K/s,  0,0055 K/s ~ 20 K/h*)
	Initialisierung.Regelventil_640_Parameter.Regelung_Sollw_Rampe_Steig_pos := 0.0055;(*Einheit: K/s,  0,0055 K/s ~ 20 K/h*)
	Initialisierung.Regelventil_640_Parameter.Stellwert_Stellung_Max := 100; (*Prozent*)
	Initialisierung.Regelventil_640_Parameter.Stellwert_Stellung_Min := 0; (*Prozent*)
	Initialisierung.Regelventil_640_Parameter.Zeit_Nachl := 15000; (*Millisekunden*)
	Initialisierung.Regelventil_640_Parameter.Zeit_Vorl := 15000; (*Millisekunden*)

	Initialisierung.Regelventil_660_Parameter.AutoQuittierung := 0;
	Initialisierung.Regelventil_660_Parameter.Regelung_PI_Kp := 0.265; (*Einheitslos*)
	Initialisierung.Regelventil_660_Parameter.Regelung_PI_Tctr := 5000; (*Millisekunden*)
	Initialisierung.Regelventil_660_Parameter.Regelung_PI_Tn := 15000; (*Millisekunden*)
	Initialisierung.Regelventil_660_Parameter.Regelung_Sollw_Max := 35; (*Grad Celsius*)
	Initialisierung.Regelventil_660_Parameter.Regelung_Sollw_Min := 5; (*Grad Celsius*)
	Initialisierung.Regelventil_660_Parameter.Regelung_Sollw_Rampe_Steig_neg := 0.0055;(*Einheit: K/s,  0,0055 K/s ~ 20 K/h*)
	Initialisierung.Regelventil_660_Parameter.Regelung_Sollw_Rampe_Steig_pos := 0.0055;(*Einheit: K/s,  0,0055 K/s ~ 20 K/h*)
	Initialisierung.Regelventil_660_Parameter.Stellwert_Stellung_Max := 100; (*Prozent*)
	Initialisierung.Regelventil_660_Parameter.Stellwert_Stellung_Min := 0; (*Prozent*)
	Initialisierung.Regelventil_660_Parameter.Zeit_Nachl := 15000; (*Millisekunden*)
	Initialisierung.Regelventil_660_Parameter.Zeit_Vorl := 15000; (*Millisekunden*)


(*Parameter System Absorptionskältemaschine *)
	Initialisierung.System_AKM_Parameter.AutoQuittierung := 0;
	Initialisierung.System_AKM_Parameter.Stellwert_Temperatur_KW_Max := 20; (*Grad Celsius*)
	Initialisierung.System_AKM_Parameter.Stellwert_Temperatur_KW_Min := 10; (*Grad Celsius*)
	Initialisierung.System_AKM_Parameter.Stellwert_Temperatur_WW_Max := 50; (*Grad Celsius*)
	Initialisierung.System_AKM_Parameter.Stellwert_Temperatur_WW_Min := 30; (*Grad Celsius*)
	Initialisierung.System_AKM_Parameter.Zeit_Nachl := 30; (*Millisekunden*)
	Initialisierung.System_AKM_Parameter.Zeit_Vorl := 30; (*Millisekunden*)



(*Parameter System Beleuchtung *)
	Initialisierung.System_Bel_Parameter.AutoQuittierung := 0;
	Initialisierung.System_Bel_Parameter.Zeit_Vorl := 1000; (* Millisekunden *)
	Initialisierung.System_Bel_Parameter.Zeit_Nachl := 1000; (* Millisekunden *)
	Initialisierung.System_Bel_Parameter.Nachtabsenkung_Uhrzeit_Stunde_Start := 23; (*Uhr*)
	Initialisierung.System_Bel_Parameter.Nachtabsenkung_Uhrzeit_Stunde_Ende := 6; (*Uhr*)

(*Parameter System Betonspeicher allgemein *)
	Initialisierung.System_BSp_Parameter.AutoQuittierung := 0;
	Initialisierung.System_BSp_Parameter.Kennlinie_Tctr := 5000; (*Millisekunden*)


(*Parameter System Betonspeicher 795 *)
	Initialisierung.Stellventil_105_Parameter.AutoQuittierung := 0;
	Initialisierung.Stellventil_105_Parameter.Zeit_Stellen0 := 35000; (*Millisekunden*)
	Initialisierung.Stellventil_105_Parameter.Zeit_Stellen1 := 20000; (*Millisekunden*)

	Initialisierung.Pumpe_105_Parameter.AutoQuittierung := 0;
	Initialisierung.Pumpe_105_Parameter.Regelung_PI_Kp := 0.265; (*Einheitslos*)
	Initialisierung.Pumpe_105_Parameter.Regelung_PI_Tctr := 5000; (*Millisekunden*)
	Initialisierung.Pumpe_105_Parameter.Regelung_PI_Tn := 15000; (*Millisekunden*)
	Initialisierung.Pumpe_105_Parameter.Stellwert_Leistung_Max := 100; (*Prozent*)
	Initialisierung.Pumpe_105_Parameter.Stellwert_Leistung_Min := 30; (*Prozent*)
	Initialisierung.Pumpe_105_Parameter.Zeit_Nachl := 2000; (*Millisekunden*)
	Initialisierung.Pumpe_105_Parameter.Zeit_Vorl := 2000; (*Millisekunden*)



(*Parameter System Betonspeicher 797 *)
	Initialisierung.Stellventil_205_Parameter.AutoQuittierung := 0;
	Initialisierung.Stellventil_205_Parameter.Zeit_Stellen0 := 35000; (*Millisekunden*)
	Initialisierung.Stellventil_205_Parameter.Zeit_Stellen1 := 20000; (*Millisekunden*)

	Initialisierung.Pumpe_205_Parameter.AutoQuittierung := 0;
	Initialisierung.Pumpe_205_Parameter.Regelung_PI_Kp := 0.265; (*Einheitslos*)
	Initialisierung.Pumpe_205_Parameter.Regelung_PI_Tctr := 5000; (*Millisekunden*)
	Initialisierung.Pumpe_205_Parameter.Regelung_PI_Tn := 15000; (*Millisekunden*)
	Initialisierung.Pumpe_205_Parameter.Stellwert_Leistung_Max := 100; (*Prozent*)
	Initialisierung.Pumpe_205_Parameter.Stellwert_Leistung_Min := 30; (*Prozent*)
	Initialisierung.Pumpe_205_Parameter.Zeit_Nachl := 2000; (*Millisekunden*)
	Initialisierung.Pumpe_205_Parameter.Zeit_Vorl := 2000; (*Millisekunden*)


(*Parameter System Blockheizkraftwerk allgemein *)
	Initialisierung.System_BHKW_Parameter.AutoQuittierung := 0;
	Initialisierung.System_BHKW_Parameter.Zeit_Vorl := T#1m; (*Minuten*)(*Zeit, nach der BHKW auch ohne Rückmeldung angeschaltet wird *)
	Initialisierung.System_BHKW_Parameter.Zeit_Nachl := T#15m; (*Minuten*)


(*Parameter System BHKW 921 *)
	Initialisierung.Anlage_BHKW_921_Parameter.AutoQuittierung := 0;
	Initialisierung.Anlage_BHKW_921_Parameter.Regelung_PI_Kp := 0.265;
	Initialisierung.Anlage_BHKW_921_Parameter.Regelung_PI_Tctr := 5000;(*Millisekunden*)
	Initialisierung.Anlage_BHKW_921_Parameter.Regelung_PI_Tn := 15;(*Millisekunden*)
	Initialisierung.Anlage_BHKW_921_Parameter.Stellwert_Leistung_Max := 100;(*Prozent*)
	Initialisierung.Anlage_BHKW_921_Parameter.Stellwert_Leistung_Min := 0;(*Prozent*)
	Initialisierung.Anlage_BHKW_921_Parameter.Temp_Ruecklauf_Max := 62; (*Grad Celsius*)
	Initialisierung.Anlage_BHKW_921_Parameter.Temp_Ruecklauf_Min := 30; (*Grad Celsius*)
	Initialisierung.Anlage_BHKW_921_Parameter.Zeit_Nachl := 900000; (*Millisekunden*)(*15 min*)
	Initialisierung.Anlage_BHKW_921_Parameter.Zeit_Vorl := 120000; (*Millisekunden*)(*120 sec *)
	Initialisierung.Anlage_BHKW_921_Parameter.Temp_Kuehlwasser_Max := 90; (*Grad Celsius*)
(*	Initialisierung.Anlage_BHKW_921_Parameter.Temp_Kuehlwasser_Max_Dauer := T#2m; (*Minuten*)*)

	Initialisierung.Stellventil_321_Parameter.AutoQuittierung := 0;
	Initialisierung.Stellventil_321_Parameter.Zeit_Stellen0 := 10000;(*Millisekunden*)
	Initialisierung.Stellventil_321_Parameter.Zeit_Stellen1 := 10000;(*Millisekunden*)

	Initialisierung.Pumpe_321_Parameter.AutoQuittierung := 0;
	Initialisierung.Pumpe_321_Parameter.Regelung_PI_Kp := 0.265;
	Initialisierung.Pumpe_321_Parameter.Regelung_PI_Tctr := 5000;(*Millisekunden*)
	Initialisierung.Pumpe_321_Parameter.Regelung_PI_Tn := 15000;(*Millisekunden*)
	Initialisierung.Pumpe_321_Parameter.Stellwert_Leistung_Max := 100;(*Prozent*)
	Initialisierung.Pumpe_321_Parameter.Stellwert_Leistung_Min := 50;(*Prozent*)
	Initialisierung.Pumpe_321_Parameter.Zeit_Nachl := 2000;(*Millisekunden*)
	Initialisierung.Pumpe_321_Parameter.Zeit_Vorl := 2000;(*Millisekunden*)

	Initialisierung.Regelventil_321_Parameter.AutoQuittierung := 0;
	Initialisierung.Regelventil_321_Parameter.Regelung_PI_Kp := 5;
	Initialisierung.Regelventil_321_Parameter.Regelung_PI_Tctr := 500;(*Millisekunden*)
	Initialisierung.Regelventil_321_Parameter.Regelung_PI_Tn := 150000;(*Millisekunden*)
	Initialisierung.Regelventil_321_Parameter.Regelung_Sollw_Max := 80;(*Grad Celsius*)
	Initialisierung.Regelventil_321_Parameter.Regelung_Sollw_Min := 40;(*Grad Celsius*)
	Initialisierung.Regelventil_321_Parameter.Regelung_Sollw_Rampe_Steig_neg := 3; (*Einheit: K/s*)
	Initialisierung.Regelventil_321_Parameter.Regelung_Sollw_Rampe_Steig_pos := 3; (*Einheit: K/s*)
	Initialisierung.Regelventil_321_Parameter.Stellwert_Stellung_Max := 100;(*Prozent*)
	Initialisierung.Regelventil_321_Parameter.Stellwert_Stellung_Min := 0;(*Prozent*)
	Initialisierung.Regelventil_321_Parameter.Zeit_Nachl := 15000;(*Millisekunden*)
	Initialisierung.Regelventil_321_Parameter.Zeit_Vorl := 15000;(*Millisekunden*)

(*Parameter System BHKW 922 *)
	Initialisierung.Anlage_BHKW_922_Parameter.AutoQuittierung := 0;
	Initialisierung.Anlage_BHKW_922_Parameter.Regelung_PI_Kp := 0.265;
	Initialisierung.Anlage_BHKW_922_Parameter.Regelung_PI_Tctr := 5000;(*Millisekunden*)
	Initialisierung.Anlage_BHKW_922_Parameter.Regelung_PI_Tn := 15;(*Millisekunden*)
	Initialisierung.Anlage_BHKW_922_Parameter.Stellwert_Leistung_Max := 100;(*Prozent*)
	Initialisierung.Anlage_BHKW_922_Parameter.Stellwert_Leistung_Min := 0;(*Prozent*)
	Initialisierung.Anlage_BHKW_922_Parameter.Temp_Ruecklauf_Max := 62; (*Grad Celsius*)
	Initialisierung.Anlage_BHKW_922_Parameter.Temp_Ruecklauf_Min := 30; (*Grad Celsius*)
	Initialisierung.Anlage_BHKW_922_Parameter.Zeit_Nachl := 900000; (*Millisekunden*)(*15 min*)
	Initialisierung.Anlage_BHKW_922_Parameter.Zeit_Vorl := 30000;(*Millisekunden*) (*30 sec *)
	Initialisierung.Anlage_BHKW_922_Parameter.Temp_Kuehlwasser_Max := 90; (*Grad Celsius*)
(*	Initialisierung.Anlage_BHKW_922_Parameter.Temp_Kuehlwasser_Max_Dauer := T#5m; (*Minuten*)*)

	Initialisierung.Stellventil_322_Parameter.AutoQuittierung := 0;
	Initialisierung.Stellventil_322_Parameter.Zeit_Stellen0 := 10000;(*Millisekunden*)
	Initialisierung.Stellventil_322_Parameter.Zeit_Stellen1 := 10000;(*Millisekunden*)

	Initialisierung.Pumpe_322_Parameter.AutoQuittierung := 0;
	Initialisierung.Pumpe_322_Parameter.Regelung_PI_Kp := 0.265;
	Initialisierung.Pumpe_322_Parameter.Regelung_PI_Tctr := 5000;(*Millisekunden*)
	Initialisierung.Pumpe_322_Parameter.Regelung_PI_Tn := 15000;(*Millisekunden*)
	Initialisierung.Pumpe_322_Parameter.Stellwert_Leistung_Max := 100;(*Prozent*)
	Initialisierung.Pumpe_322_Parameter.Stellwert_Leistung_Min := 50;(*Prozent*)
	Initialisierung.Pumpe_322_Parameter.Zeit_Nachl := 2000;(*Millisekunden*)
	Initialisierung.Pumpe_322_Parameter.Zeit_Vorl := 2000;(*Millisekunden*)

	Initialisierung.Regelventil_322_Parameter.AutoQuittierung := 0;
	Initialisierung.Regelventil_322_Parameter.Regelung_PI_Kp := 5;
	Initialisierung.Regelventil_322_Parameter.Regelung_PI_Tctr := 500;(*Millisekunden*)
	Initialisierung.Regelventil_322_Parameter.Regelung_PI_Tn := 150000;(*Millisekunden*)
	Initialisierung.Regelventil_322_Parameter.Regelung_Sollw_Max := 80;(*Grad Celsius*)
	Initialisierung.Regelventil_322_Parameter.Regelung_Sollw_Min := 40;(*Grad Celsius*)
	Initialisierung.Regelventil_322_Parameter.Regelung_Sollw_Rampe_Steig_neg := 3; (*Einheit: K/s*)
	Initialisierung.Regelventil_322_Parameter.Regelung_Sollw_Rampe_Steig_pos := 3; (*Einheit: K/s*)
	Initialisierung.Regelventil_322_Parameter.Stellwert_Stellung_Max := 100;(*Prozent*)
	Initialisierung.Regelventil_322_Parameter.Stellwert_Stellung_Min := 0;(*Prozent*)
	Initialisierung.Regelventil_322_Parameter.Zeit_Nachl := 15000;(*Millisekunden*)
	Initialisierung.Regelventil_322_Parameter.Zeit_Vorl := 15000;(*Millisekunden*)

(*Parameter System Brennwertkessel *)
	Initialisierung.System_BWK_Parameter.AutoQuittierung := 0;

	Initialisierung.Stellventil_331_Parameter.AutoQuittierung := 0;
	Initialisierung.Stellventil_331_Parameter.Zeit_Stellen0 := 10000;(*Millisekunden*)
	Initialisierung.Stellventil_331_Parameter.Zeit_Stellen1 := 10000;(*Millisekunden*)

	Initialisierung.Anlage_BWK_Parameter.AutoQuittierung := 0;
	Initialisierung.Anlage_BWK_Parameter.Stellwert_Leistung_Max := 100;
	Initialisierung.Anlage_BWK_Parameter.Stellwert_Leistung_Min := 0;
	Initialisierung.Anlage_BWK_Parameter.Stellwert_Temperatur_Max := 100; (*Grad Celsius*)
	Initialisierung.Anlage_BWK_Parameter.Stellwert_Temperatur_Min := 30; (*Grad Celsius*)
	Initialisierung.Anlage_BWK_Parameter.Temp_Ruecklauf_Max := 85; (*Grad Celsius*)
	Initialisierung.Anlage_BWK_Parameter.Temp_Ruecklauf_Min := 30; (*Grad Celsius*)
	Initialisierung.Anlage_BWK_Parameter.Zeit_Nachl := 300000; (*Millisekunden*)(*5 min -> geändert von 15 min MLi 29.04.21*)
	Initialisierung.Anlage_BWK_Parameter.Zeit_Vorl := 60000;(*Millisekunden*)

	Initialisierung.Regelventil_331_Parameter.AutoQuittierung := 0;
	Initialisierung.Regelventil_331_Parameter.Regelung_PI_Kp := 0.5;
	Initialisierung.Regelventil_331_Parameter.Regelung_PI_Tctr := 5000;(*Millisekunden*)
	Initialisierung.Regelventil_331_Parameter.Regelung_PI_Tn := 15000;(*Millisekunden*)
	Initialisierung.Regelventil_331_Parameter.Regelung_Sollw_Max := 45;(*Grad Celsius*)
	Initialisierung.Regelventil_331_Parameter.Regelung_Sollw_Min := 15;(*Grad Celsius*)
	Initialisierung.Regelventil_331_Parameter.Regelung_Sollw_Rampe_Steig_neg := 0.003; (*Einheit: K/s,  0,003 K/s ~ 10 K/h*)
	Initialisierung.Regelventil_331_Parameter.Regelung_Sollw_Rampe_Steig_pos := 0.003; (*Einheit: K/s*)
	Initialisierung.Regelventil_331_Parameter.Stellwert_Stellung_Max := 100;(*Prozent*)
	Initialisierung.Regelventil_331_Parameter.Stellwert_Stellung_Min := 0;(*Prozent*)
	Initialisierung.Regelventil_331_Parameter.Zeit_Nachl := 15000;(*Millisekunden*)
	Initialisierung.Regelventil_331_Parameter.Zeit_Vorl := 15000;(*Millisekunden*)

(*Parameter System Druckluftkompressor *)
	Initialisierung.System_DLK_Parameter.AutoQuittierung := 0;

	Initialisierung.Stellventil_251_Parameter.AutoQuittierung := 0;
	Initialisierung.Stellventil_251_Parameter.Zeit_Stellen0 := 10000;(*Millisekunden*)
	Initialisierung.Stellventil_251_Parameter.Zeit_Stellen1 := 10000;(*Millisekunden*)

	Initialisierung.Pumpe_251_Parameter.AutoQuittierung := 0;
	Initialisierung.Pumpe_251_Parameter.Regelung_PI_Kp := 0.265;
	Initialisierung.Pumpe_251_Parameter.Regelung_PI_Tctr := 5000;(*Millisekunden*)
	Initialisierung.Pumpe_251_Parameter.Regelung_PI_Tn := 15000;(*Millisekunden*)
	Initialisierung.Pumpe_251_Parameter.Stellwert_Leistung_Max := 100;(*Prozent*)
	Initialisierung.Pumpe_251_Parameter.Stellwert_Leistung_Min := 50;(*Prozent*)
	Initialisierung.Pumpe_251_Parameter.Zeit_Nachl := 2000;(*Millisekunden*)
	Initialisierung.Pumpe_251_Parameter.Zeit_Vorl := 2000;(*Millisekunden*)

	Initialisierung.Regelventil_251_Parameter.AutoQuittierung := 0;
	Initialisierung.Regelventil_251_Parameter.Regelung_PI_Kp := 5;
	Initialisierung.Regelventil_251_Parameter.Regelung_PI_Tctr := 500;(*Millisekunden*)
	Initialisierung.Regelventil_251_Parameter.Regelung_PI_Tn := 150000;(*Millisekunden*)
	Initialisierung.Regelventil_251_Parameter.Regelung_Sollw_Max := 60;(*Grad Celsius*)
	Initialisierung.Regelventil_251_Parameter.Regelung_Sollw_Min := 15;(*Grad Celsius*)
	Initialisierung.Regelventil_251_Parameter.Regelung_Sollw_Rampe_Steig_neg := 3; (*Einheit: K/s*)
	Initialisierung.Regelventil_251_Parameter.Regelung_Sollw_Rampe_Steig_pos := 3; (*Einheit: K/s*)
	Initialisierung.Regelventil_251_Parameter.Stellwert_Stellung_Max := 100;(*Prozent*)
	Initialisierung.Regelventil_251_Parameter.Stellwert_Stellung_Min := 0;(*Prozent*)
	Initialisierung.Regelventil_251_Parameter.Zeit_Nachl := 15000;(*Millisekunden*)
	Initialisierung.Regelventil_251_Parameter.Zeit_Vorl := 15000;(*Millisekunden*)

(* Parameter Anlage Druckluftkompressor *)
	Initialisierung.Anlage_DLK_Parameter.AutoQuittierung := 0;
	Initialisierung.Anlage_DLK_Parameter.Temp_Warmwasser_Max := 45; (*Grad Celsius*)

(*Parameter System Fenster *)

	Initialisierung.Fenster_Halle_OST_Parameter.AutoQuittierung := 0;
	Initialisierung.Fenster_Halle_OST_Parameter.Zeit_Stellen0 := 120000;(*Millisekunden*)
	Initialisierung.Fenster_Halle_OST_Parameter.Zeit_Stellen1 := 120000;(*Millisekunden*)

	Initialisierung.Fenster_Halle_WEST_Parameter.AutoQuittierung := 0;
	Initialisierung.Fenster_Halle_WEST_Parameter.Zeit_Stellen0 := 120000;(*Millisekunden*)
	Initialisierung.Fenster_Halle_WEST_Parameter.Zeit_Stellen1 := 120000;(*Millisekunden*)

(*Parameter System Fußbodentemperierung *)

	Initialisierung.System_FBT_Parameter.Temp_Warmwasser_Max := 45; (*Grad Celsius*)
	Initialisierung.System_FBT_Parameter.Temp_Warmwasser_Min := 35; (*Grad Celsius*)
	Initialisierung.System_FBT_Parameter.Temp_Kaltwasser_Max := 20; (*Grad Celsius*)
	Initialisierung.System_FBT_Parameter.Temp_Kaltwasser_Min := 12 ; (*Grad Celsius*)

	Initialisierung.System_FBT_Parameter.Temp_Vorl_Max := 45;
	Initialisierung.System_FBT_Parameter.Temp_Vorl_Min := 5;
	(* Heizkurve mit Neigung 0.6 https://www.vaillant.de/heizung/heizung-verstehen/tipps-rund-um-ihre-heizung/vorlauf-rucklauftemperatur/*)
	Initialisierung.System_FBT_Parameter.Kennlinie_Heizung.Temp_Aussen_Max := 15; (*Grad Celsius*)
	Initialisierung.System_FBT_Parameter.Kennlinie_Heizung.Temp_Aussen_Min := -12; (*Grad Celsius*)
	Initialisierung.System_FBT_Parameter.Kennlinie_Heizung.Temp_Vorl_Max := 43; (*Grad Celsius*)
	Initialisierung.System_FBT_Parameter.Kennlinie_Heizung.Temp_Vorl_Min := 25; (*Grad Celsius*)
	Initialisierung.System_FBT_Parameter.Kennlinie_Kuehlung.Temp_Aussen_Max := 28; (*Grad Celsius*)
	Initialisierung.System_FBT_Parameter.Kennlinie_Kuehlung.Temp_Aussen_Min := 16; (*Grad Celsius*)
	Initialisierung.System_FBT_Parameter.Kennlinie_Kuehlung.Temp_Vorl_Max := 18; (*Grad Celsius*)
	Initialisierung.System_FBT_Parameter.Kennlinie_Kuehlung.Temp_Vorl_Min := 16; (*Grad Celsius*)

	Initialisierung.System_FBT_Parameter.Nachtabsenkung_Mo.Temp_Absenkung := 10; (*Grad Celsius*)
	Initialisierung.System_FBT_Parameter.Nachtabsenkung_Mo.Uhrzeit_Stunde_Start := 21;(*Uhr*)
	Initialisierung.System_FBT_Parameter.Nachtabsenkung_Mo.Uhrzeit_Stunde_Ende := 3.5;(*Uhr*)
	Initialisierung.System_FBT_Parameter.Nachtabsenkung_Di.Temp_Absenkung := 10; (*Grad Celsius*)
	Initialisierung.System_FBT_Parameter.Nachtabsenkung_Di.Uhrzeit_Stunde_Start := 21;(*Uhr*)
	Initialisierung.System_FBT_Parameter.Nachtabsenkung_Di.Uhrzeit_Stunde_Ende := 3.5;(*Uhr*)
	Initialisierung.System_FBT_Parameter.Nachtabsenkung_Mi.Temp_Absenkung := 10; (*Grad Celsius*)
	Initialisierung.System_FBT_Parameter.Nachtabsenkung_Mi.Uhrzeit_Stunde_Start := 21;(*Uhr*)
	Initialisierung.System_FBT_Parameter.Nachtabsenkung_Mi.Uhrzeit_Stunde_Ende := 3.5;(*Uhr*)
	Initialisierung.System_FBT_Parameter.Nachtabsenkung_Do.Temp_Absenkung := 10; (*Grad Celsius*)
	Initialisierung.System_FBT_Parameter.Nachtabsenkung_Do.Uhrzeit_Stunde_Start := 21;(*Uhr*)
	Initialisierung.System_FBT_Parameter.Nachtabsenkung_Do.Uhrzeit_Stunde_Ende := 3.5;(*Uhr*)
	Initialisierung.System_FBT_Parameter.Nachtabsenkung_Fr.Temp_Absenkung := 10; (*Grad Celsius*)
	Initialisierung.System_FBT_Parameter.Nachtabsenkung_Fr.Uhrzeit_Stunde_Start := 21;(*Uhr*)
	Initialisierung.System_FBT_Parameter.Nachtabsenkung_Fr.Uhrzeit_Stunde_Ende := 3.5;(*Uhr*)
	Initialisierung.System_FBT_Parameter.Nachtabsenkung_Sa.Temp_Absenkung := 10; (*Grad Celsius*)
	Initialisierung.System_FBT_Parameter.Nachtabsenkung_Sa.Uhrzeit_Stunde_Start := 21;(*Uhr*)
	Initialisierung.System_FBT_Parameter.Nachtabsenkung_Sa.Uhrzeit_Stunde_Ende := 3.5;(*Uhr*)
	Initialisierung.System_FBT_Parameter.Nachtabsenkung_So.Temp_Absenkung := 10; (*Grad Celsius*)
	Initialisierung.System_FBT_Parameter.Nachtabsenkung_So.Uhrzeit_Stunde_Start := 21;(*Uhr*)
	Initialisierung.System_FBT_Parameter.Nachtabsenkung_So.Uhrzeit_Stunde_Ende := 3.5;(*Uhr*)

	Initialisierung.Stellventil_423_Parameter.AutoQuittierung := 0;
	Initialisierung.Stellventil_423_Parameter.Zeit_Stellen0 := 10000;(*Millisekunden*)
	Initialisierung.Stellventil_423_Parameter.Zeit_Stellen1 := 10000;(*Millisekunden*)

	Initialisierung.Stellventil_424_Parameter.AutoQuittierung := 0;
	Initialisierung.Stellventil_424_Parameter.Zeit_Stellen0 := 10000;(*Millisekunden*)
	Initialisierung.Stellventil_424_Parameter.Zeit_Stellen1 := 10000;(*Millisekunden*)

	Initialisierung.Regelventil_425_Parameter.AutoQuittierung := 0;
	Initialisierung.Regelventil_425_Parameter.Regelung_PI_Kp := 0.5;
	Initialisierung.Regelventil_425_Parameter.Regelung_PI_Tctr := 5000;(*Millisekunden*)
	Initialisierung.Regelventil_425_Parameter.Regelung_PI_Tn := 15000;(*Millisekunden*)
	Initialisierung.Regelventil_425_Parameter.Regelung_Sollw_Max := 45;(*Grad Celsius*)
	Initialisierung.Regelventil_425_Parameter.Regelung_Sollw_Min := 15;(*Grad Celsius*)
	Initialisierung.Regelventil_425_Parameter.Regelung_Sollw_Rampe_Steig_neg := 0.003; (*Einheit: K/s,  0,003 K/s ~ 10 K/h*)
	Initialisierung.Regelventil_425_Parameter.Regelung_Sollw_Rampe_Steig_pos := 0.003; (*Einheit: K/s*)
	Initialisierung.Regelventil_425_Parameter.Stellwert_Stellung_Max := 100;(*Prozent*)
	Initialisierung.Regelventil_425_Parameter.Stellwert_Stellung_Min := 0;(*Prozent*)
	Initialisierung.Regelventil_425_Parameter.Zeit_Nachl := 15000;(*Millisekunden*)
	Initialisierung.Regelventil_425_Parameter.Zeit_Vorl := 15000;(*Millisekunden*)

	Initialisierung.Pumpe_425_Parameter.AutoQuittierung := 0;
	Initialisierung.Pumpe_425_Parameter.Regelung_PI_Kp := 0.4;
	Initialisierung.Pumpe_425_Parameter.Regelung_PI_Tctr := 5000;(*Millisekunden*)
	Initialisierung.Pumpe_425_Parameter.Regelung_PI_Tn := 15000;(*Millisekunden*)
	Initialisierung.Pumpe_425_Parameter.Stellwert_Leistung_Max := 100;(*Prozent*)
	Initialisierung.Pumpe_425_Parameter.Stellwert_Leistung_Min := 50;(*Prozent*)
	Initialisierung.Pumpe_425_Parameter.Zeit_Nachl := 2000;(*Millisekunden*)
	Initialisierung.Pumpe_425_Parameter.Zeit_Vorl := 2000;(*Millisekunden*)


(*Parameter System Hybrider Energiespeicher *)
	Initialisierung.System_HES_Parameter.AutoQuittierung := 0;

	Initialisierung.Anlage_HES_Parameter.Temp_Kuehlwasser_Max := 17; (*Grad Celsius*)
	Initialisierung.Anlage_HES_Parameter.Temp_Kuehlwasser_Min := 12; (*Grad Celsius*)
	Initialisierung.Anlage_HES_Parameter.AutoQuittierung := 0;

	Initialisierung.Stellventil_191_Parameter.AutoQuittierung := 0;
	Initialisierung.Stellventil_191_Parameter.Zeit_Stellen0 := 10000;(*Millisekunden*)
	Initialisierung.Stellventil_191_Parameter.Zeit_Stellen1 := 10000;(*Millisekunden*)

	Initialisierung.Pumpe_191_Parameter.AutoQuittierung := 0;
	Initialisierung.Pumpe_191_Parameter.Regelung_PI_Kp := 0.265;
	Initialisierung.Pumpe_191_Parameter.Regelung_PI_Tctr := 5000;(*Millisekunden*)
	Initialisierung.Pumpe_191_Parameter.Regelung_PI_Tn := 15000;(*Millisekunden*)
	Initialisierung.Pumpe_191_Parameter.Stellwert_Leistung_Max := 100;(*Prozent*)
	Initialisierung.Pumpe_191_Parameter.Stellwert_Leistung_Min := 30;(*Prozent*)
	Initialisierung.Pumpe_191_Parameter.Zeit_Nachl := 2000;(*Millisekunden*)
	Initialisierung.Pumpe_191_Parameter.Zeit_Vorl := 2000;(*Millisekunden*)


(*Parameter System Härteofen Heißwasser *)
	Initialisierung.System_HOHW_Parameter.AutoQuittierung := 0;

	Initialisierung.Anlage_HO_Parameter.Temp_Heisswasser_Max := 85; (*Grad Celsius*)
	Initialisierung.Anlage_HO_Parameter.Temp_Warmwasser:= 35; (*Grad Celsius*)
	Initialisierung.Anlage_HO_Parameter.Temp_Warmwasser_Max := 60; (*Grad Celsius*)

	Initialisierung.Stellventil_361_Parameter.AutoQuittierung := 0;
	Initialisierung.Stellventil_361_Parameter.Zeit_Stellen0 := 10000;(*Millisekunden*)
	Initialisierung.Stellventil_361_Parameter.Zeit_Stellen1 := 10000;(*Millisekunden*)

	Initialisierung.Pumpe_361_Parameter.AutoQuittierung := 0;
	Initialisierung.Pumpe_361_Parameter.Regelung_PI_Kp := 0.265;
	Initialisierung.Pumpe_361_Parameter.Regelung_PI_Tctr := 5000;(*Millisekunden*)
	Initialisierung.Pumpe_361_Parameter.Regelung_PI_Tn := 15000;(*Millisekunden*)
	Initialisierung.Pumpe_361_Parameter.Stellwert_Leistung_Max := 100;(*Prozent*)
	Initialisierung.Pumpe_361_Parameter.Stellwert_Leistung_Min := 30;(*Prozent*)
	Initialisierung.Pumpe_361_Parameter.Zeit_Nachl := 2000;(*Millisekunden*)
	Initialisierung.Pumpe_361_Parameter.Zeit_Vorl := 2000;(*Millisekunden*)

	Initialisierung.Regelventil_361_Parameter.AutoQuittierung := 0;
	Initialisierung.Regelventil_361_Parameter.Regelung_PI_Kp := 0.265;
	Initialisierung.Regelventil_361_Parameter.Regelung_PI_Tctr := 5000;(*Millisekunden*)
	Initialisierung.Regelventil_361_Parameter.Regelung_PI_Tn := 15000;(*Millisekunden*)
	Initialisierung.Regelventil_361_Parameter.Regelung_Sollw_Max := 35; (*Grad Celsius*)
	Initialisierung.Regelventil_361_Parameter.Regelung_Sollw_Min := 15; (*Grad Celsius*)
	Initialisierung.Regelventil_361_Parameter.Regelung_Sollw_Rampe_Steig_neg := 0.0005;(*Einheit: K/s,  0,0005 K/s ~ 2 K/h*)
	Initialisierung.Regelventil_361_Parameter.Regelung_Sollw_Rampe_Steig_pos := 0.0005;(*Einheit: K/s,  0,0005 K/s ~ 2 K/h*)
	Initialisierung.Regelventil_361_Parameter.Stellwert_Stellung_Max := 100;(*Prozent*)
	Initialisierung.Regelventil_361_Parameter.Stellwert_Stellung_Min := 0;(*Prozent*)
	Initialisierung.Regelventil_361_Parameter.Zeit_Nachl := 15000;(*Millisekunden*)
	Initialisierung.Regelventil_361_Parameter.Zeit_Vorl := 15000;(*Millisekunden*)

(*Parameter System Härteofen Warmwasser *)
	Initialisierung.System_HOWW_Parameter.AutoQuittierung := 0;

	Initialisierung.Stellventil_261_Parameter.AutoQuittierung := 0;
	Initialisierung.Stellventil_261_Parameter.Zeit_Stellen0 := 10000;(*Millisekunden*)
	Initialisierung.Stellventil_261_Parameter.Zeit_Stellen1 := 10000;(*Millisekunden*)

	Initialisierung.Pumpe_261_Parameter.AutoQuittierung := 0;
	Initialisierung.Pumpe_261_Parameter.Regelung_PI_Kp := 0.265;
	Initialisierung.Pumpe_261_Parameter.Regelung_PI_Tctr := 5000;(*Millisekunden*)
	Initialisierung.Pumpe_261_Parameter.Regelung_PI_Tn := 15000;(*Millisekunden*)
	Initialisierung.Pumpe_261_Parameter.Stellwert_Leistung_Max := 100;(*Prozent*)
	Initialisierung.Pumpe_261_Parameter.Stellwert_Leistung_Min := 30;(*Prozent*)
	Initialisierung.Pumpe_261_Parameter.Zeit_Nachl := 2000;(*Millisekunden*)
	Initialisierung.Pumpe_261_Parameter.Zeit_Vorl := 2000;(*Millisekunden*)

	Initialisierung.Regelventil_261_Parameter.AutoQuittierung := 0;
	Initialisierung.Regelventil_261_Parameter.Regelung_PI_Kp := 0.265;
	Initialisierung.Regelventil_261_Parameter.Regelung_PI_Tctr := 5000;(*Millisekunden*)
	Initialisierung.Regelventil_261_Parameter.Regelung_PI_Tn := 15000;(*Millisekunden*)
	Initialisierung.Regelventil_261_Parameter.Regelung_Sollw_Max := 35; (*Grad Celsius*)
	Initialisierung.Regelventil_261_Parameter.Regelung_Sollw_Min := 15; (*Grad Celsius*)
	Initialisierung.Regelventil_261_Parameter.Regelung_Sollw_Rampe_Steig_neg := 0.0005;(*Einheit: K/s,  0,0005 K/s ~ 2 K/h*)
	Initialisierung.Regelventil_261_Parameter.Regelung_Sollw_Rampe_Steig_pos := 0.0005;(*Einheit: K/s,  0,0005 K/s ~ 2 K/h*)
	Initialisierung.Regelventil_261_Parameter.Stellwert_Stellung_Max := 100;(*Prozent*)
	Initialisierung.Regelventil_261_Parameter.Stellwert_Stellung_Min := 0;(*Prozent*)
	Initialisierung.Regelventil_261_Parameter.Zeit_Nachl := 15000;(*Millisekunden*)
	Initialisierung.Regelventil_261_Parameter.Zeit_Vorl := 15000;(*Millisekunden*)

(*Parameter System Heizstaebe *)
	Initialisierung.System_HS_Parameter.AutoQuittierung := 0;
	Initialisierung.System_HS_Parameter.Kennlinie_Tctr := 5000;(*Millisekunden*)
	Initialisierung.System_HS_Parameter.Temp_Spreizung := 2; (*Grad Celsius*)


(*Parameter System Kältekompressor Kaltwasser *)
	Initialisierung.System_KKKW_Parameter.AutoQuittierung := 0;

	Initialisierung.Stellventil_145_Parameter.AutoQuittierung := 0;
	Initialisierung.Stellventil_145_Parameter.Zeit_Stellen0 := 35000;(*Millisekunden*)
	Initialisierung.Stellventil_145_Parameter.Zeit_Stellen1 := 10000;(*Millisekunden*)

	Initialisierung.Pumpe_145_Parameter.AutoQuittierung := 0;
	Initialisierung.Pumpe_145_Parameter.Regelung_PI_Kp := 0.265;
	Initialisierung.Pumpe_145_Parameter.Regelung_PI_Tctr := 5000;(*Millisekunden*)
	Initialisierung.Pumpe_145_Parameter.Regelung_PI_Tn := 15000;(*Millisekunden*)
	Initialisierung.Pumpe_145_Parameter.Stellwert_Leistung_Max := 100;(*Prozent*)
	Initialisierung.Pumpe_145_Parameter.Stellwert_Leistung_Min := 30;(*Prozent*)
	Initialisierung.Pumpe_145_Parameter.Zeit_Nachl := 2000;(*Millisekunden*)
	Initialisierung.Pumpe_145_Parameter.Zeit_Vorl := 2000;(*Millisekunden*)

(*Parameter System Maschinenversorgung Warmwasser *)
	Initialisierung.System_MVWW_Parameter.AutoQuittierung := 0;

	Initialisierung.System_MVWW_Parameter.Temp_Warmwasser:= 42; (*Grad Celsius*)
	Initialisierung.System_MVWW_Parameter.Temp_Warmwasser_Max := 47; (*Grad Celsius*)

	Initialisierung.Stellventil_245_Parameter.AutoQuittierung := 0;
	Initialisierung.Stellventil_245_Parameter.Zeit_Stellen0 := 35000;(*Millisekunden*)
	Initialisierung.Stellventil_245_Parameter.Zeit_Stellen1 := 10000;(*Millisekunden*)

	Initialisierung.Pumpe_245_Parameter.AutoQuittierung := 0;
	Initialisierung.Pumpe_245_Parameter.Regelung_PI_Kp := 0.265;
	Initialisierung.Pumpe_245_Parameter.Regelung_PI_Tctr := 5000;(*Millisekunden*)
	Initialisierung.Pumpe_245_Parameter.Regelung_PI_Tn := 15000;(*Millisekunden*)
	Initialisierung.Pumpe_245_Parameter.Stellwert_Leistung_Max := 100;(*Prozent*)
	Initialisierung.Pumpe_245_Parameter.Stellwert_Leistung_Min := 30;(*Prozent*)
	Initialisierung.Pumpe_245_Parameter.Zeit_Nachl := 2000;(*Millisekunden*)
	Initialisierung.Pumpe_245_Parameter.Zeit_Vorl := 2000;(*Millisekunden*)



(*Parameter System Lüftungsanlage *)
	Initialisierung.System_LA_Parameter.AutoQuittierung := 0;
	Initialisierung.System_LA_Parameter.Temp_Heisswasser_Max := 90 ; (*Grad Celsius*)
	Initialisierung.System_LA_Parameter.Temp_Heisswasser_Min := 45 ; (*Grad Celsius*)
	Initialisierung.System_LA_Parameter.Temp_Kaltwasser_Max := 25 ; (*Grad Celsius*)
	Initialisierung.System_LA_Parameter.Temp_Kaltwasser_Min := 8 ; (*Grad Celsius*)

	Initialisierung.Stellventil_453_Parameter.AutoQuittierung := 0;
	Initialisierung.Stellventil_453_Parameter.Zeit_Stellen0 := 10000;(*Millisekunden*)
	Initialisierung.Stellventil_453_Parameter.Zeit_Stellen1 := 10000;(*Millisekunden*)

	Initialisierung.Stellventil_454_Parameter.AutoQuittierung := 0;
	Initialisierung.Stellventil_454_Parameter.Zeit_Stellen0 := 10000;(*Millisekunden*)
	Initialisierung.Stellventil_454_Parameter.Zeit_Stellen1 := 10000;(*Millisekunden*)

	(*Parameter Anlage Lüftungsanlage *)
	Initialisierung.Anlage_LA_Parameter.Temp_Kuehlwasser_Max := 45; (*Grad Celsius*)
	Initialisierung.Anlage_LA_Parameter.Temp_Kuehlwasser_Min := 20; (*Grad Celsius*)
	Initialisierung.Anlage_LA_Parameter.Abluefter_Druck_Sollwert := 100; (*Prozent*)
	Initialisierung.Anlage_LA_Parameter.Ausschaltverz_Anlage_nach_Taster := 480;(*Millisekunden*)
	Initialisierung.Anlage_LA_Parameter.AutoQuittierung := 0;
	Initialisierung.Anlage_LA_Parameter.Betriebsartenschalter_Anlage := 9;
	Initialisierung.Anlage_LA_Parameter.Freie_Nachtkuehlung_AT_Grenzwert := 15; (*Grad Celsius*)
	Initialisierung.Anlage_LA_Parameter.Freie_Nachtkuehlung_Diff_AT_zu_RT_Grenzwert := 3; (*Grad Celsius*)
	Initialisierung.Anlage_LA_Parameter.Freie_Nachtkuehlung_Nacht_Raumsollwert := 22; (*Grad Celsius*)
	Initialisierung.Anlage_LA_Parameter.Seminarraum_CO2_Sollwert_bei_Lueftungsbetrieb := 1000; (*ppm?*)
	Initialisierung.Anlage_LA_Parameter.Seminarraum_Grenzwert_CO2_Lueftung_Aus := 900; (*ppm*)
	Initialisierung.Anlage_LA_Parameter.Seminarraum_Grenzwert_CO2_Lueftung_Ein := 1200; (*ppm*)
	Initialisierung.Anlage_LA_Parameter.Sollwertschiebung_Anlage_Max_AT_Sollwert := 32; (*Grad Celsius*)
	Initialisierung.Anlage_LA_Parameter.Sollwertschiebung_Anlage_Max_Sollwert := 26; (*Grad Celsius*)
	Initialisierung.Anlage_LA_Parameter.Sollwertschiebung_Anlage_Min_AT_Sollwert := 18; (*Grad Celsius*)
	Initialisierung.Anlage_LA_Parameter.Sollwertschiebung_Anlage_Min_Sollwert := 22; (*Grad Celsius*)
	Initialisierung.Anlage_LA_Parameter.Zuluefter_Drucksollwert := 350; (* mbar *)


(*Parameter System Maschinenversorgung Heißwasser *)
	Initialisierung.System_MVHW_Parameter.AutoQuittierung := 0;

	Initialisierung.Anlage_MVHW_Parameter.Temp_Heisswasser     := 75; (*Grad Celsius*)
	Initialisierung.Anlage_MVHW_Parameter.Temp_Heisswasser_Max := 90; (*Grad Celsius*)
	Initialisierung.Anlage_MVHW_Parameter.Temp_Heisswasser_Min := 60; (*Grad Celsius*)

	Initialisierung.Stellventil_300_Parameter.AutoQuittierung := 0;
	Initialisierung.Stellventil_300_Parameter.Zeit_Stellen0 := 10000;(*Millisekunden*)
	Initialisierung.Stellventil_300_Parameter.Zeit_Stellen1 := 10000;(*Millisekunden*)

	Initialisierung.Pumpe_300_Parameter.AutoQuittierung := 0;
	Initialisierung.Pumpe_300_Parameter.Regelung_PI_Kp := 0.265;
	Initialisierung.Pumpe_300_Parameter.Regelung_PI_Tctr := 5000;(*Millisekunden*)
	Initialisierung.Pumpe_300_Parameter.Regelung_PI_Tn := 15000;(*Millisekunden*)
	Initialisierung.Pumpe_300_Parameter.Stellwert_Leistung_Max := 100;(*Prozent*)
	Initialisierung.Pumpe_300_Parameter.Stellwert_Leistung_Min := 30;(*Prozent*)
	Initialisierung.Pumpe_300_Parameter.Zeit_Nachl := 2000;(*Millisekunden*)
	Initialisierung.Pumpe_300_Parameter.Zeit_Vorl := 2000;(*Millisekunden*)


(*Parameter System Maschinenversorgung Kaltwasser *)
	Initialisierung.System_MVKW_Parameter.AutoQuittierung := 0;

	Initialisierung.Anlage_MVKW_Parameter.Temp_Kaltwasser := 14; (*Grad Celsius*)
	Initialisierung.Anlage_MVKW_Parameter.Temp_Kaltwasser_Max := 20; (*Grad Celsius*)
	Initialisierung.Anlage_MVKW_Parameter.Temp_Kaltwasser_Min := 10; (*Grad Celsius*)

	Initialisierung.Stellventil_100_Parameter.AutoQuittierung := 0;
	Initialisierung.Stellventil_100_Parameter.Zeit_Stellen0 := 10000;(*Millisekunden*)
	Initialisierung.Stellventil_100_Parameter.Zeit_Stellen1 := 10000;(*Millisekunden*)

	Initialisierung.Pumpe_100_Parameter.AutoQuittierung := 0;
	Initialisierung.Pumpe_100_Parameter.Regelung_PI_Kp := 0.265;
	Initialisierung.Pumpe_100_Parameter.Regelung_PI_Tctr := 5000;(*Millisekunden*)
	Initialisierung.Pumpe_100_Parameter.Regelung_PI_Tn := 15000;(*Millisekunden*)
	Initialisierung.Pumpe_100_Parameter.Stellwert_Leistung_Max := 100;(*Prozent*)
	Initialisierung.Pumpe_100_Parameter.Stellwert_Leistung_Min := 30;(*Prozent*)
	Initialisierung.Pumpe_100_Parameter.Zeit_Nachl := 2000;(*Millisekunden*)
	Initialisierung.Pumpe_100_Parameter.Zeit_Vorl := 2000;(*Millisekunden*)





(*Parameter System Statische Heizung *)
	Initialisierung.System_SHZ_Parameter.Kennlinie_Heizung.Temp_Aussen_Max:= 15; (*Grad Celsius*)
	Initialisierung.System_SHZ_Parameter.Kennlinie_Heizung.Temp_Aussen_Min := -15; (*Grad Celsius*)
	Initialisierung.System_SHZ_Parameter.Kennlinie_Heizung.Temp_Vorl_Max := 65; (*Grad Celsius*)
	Initialisierung.System_SHZ_Parameter.Kennlinie_Heizung.Temp_Vorl_Min := 30; (*Grad Celsius*)

	Initialisierung.System_SHZ_Parameter.Temp_Heisswasser_Max := 65 ; (*Grad Celsius*)
	Initialisierung.System_SHZ_Parameter.Temp_Heisswasser_Min := 30 ; (*Grad Celsius*)

	Initialisierung.System_SHZ_Parameter.Nachtabsenkung_Mo.Temp_Absenkung := 10; (*Grad Celsius*)
	Initialisierung.System_SHZ_Parameter.Nachtabsenkung_Mo.Uhrzeit_Stunde_Start := 21;(*Uhr*)
	Initialisierung.System_SHZ_Parameter.Nachtabsenkung_Mo.Uhrzeit_Stunde_Ende := 3.5;(*Uhr*)
	Initialisierung.System_SHZ_Parameter.Nachtabsenkung_Di.Temp_Absenkung := 10; (*Grad Celsius*)
	Initialisierung.System_SHZ_Parameter.Nachtabsenkung_Di.Uhrzeit_Stunde_Start := 21;(*Uhr*)
	Initialisierung.System_SHZ_Parameter.Nachtabsenkung_Di.Uhrzeit_Stunde_Ende := 3.5;(*Uhr*)
	Initialisierung.System_SHZ_Parameter.Nachtabsenkung_Mi.Temp_Absenkung := 10; (*Grad Celsius*)
	Initialisierung.System_SHZ_Parameter.Nachtabsenkung_Mi.Uhrzeit_Stunde_Start := 21;(*Uhr*)
	Initialisierung.System_SHZ_Parameter.Nachtabsenkung_Mi.Uhrzeit_Stunde_Ende := 3.5;(*Uhr*)
	Initialisierung.System_SHZ_Parameter.Nachtabsenkung_Do.Temp_Absenkung := 10; (*Grad Celsius*)
	Initialisierung.System_SHZ_Parameter.Nachtabsenkung_Do.Uhrzeit_Stunde_Start := 21;(*Uhr*)
	Initialisierung.System_SHZ_Parameter.Nachtabsenkung_Do.Uhrzeit_Stunde_Ende := 3.5;(*Uhr*)
	Initialisierung.System_SHZ_Parameter.Nachtabsenkung_Fr.Temp_Absenkung := 10; (*Grad Celsius*)
	Initialisierung.System_SHZ_Parameter.Nachtabsenkung_Fr.Uhrzeit_Stunde_Start := 21;(*Uhr*)
	Initialisierung.System_SHZ_Parameter.Nachtabsenkung_Fr.Uhrzeit_Stunde_Ende := 3.5;(*Uhr*)
	Initialisierung.System_SHZ_Parameter.Nachtabsenkung_Sa.Temp_Absenkung := 10; (*Grad Celsius*)
	Initialisierung.System_SHZ_Parameter.Nachtabsenkung_Sa.Uhrzeit_Stunde_Start := 21;(*Uhr*)
	Initialisierung.System_SHZ_Parameter.Nachtabsenkung_Sa.Uhrzeit_Stunde_Ende := 3.5;(*Uhr*)
	Initialisierung.System_SHZ_Parameter.Nachtabsenkung_So.Temp_Absenkung := 10; (*Grad Celsius*)
	Initialisierung.System_SHZ_Parameter.Nachtabsenkung_So.Uhrzeit_Stunde_Start := 21;(*Uhr*)
	Initialisierung.System_SHZ_Parameter.Nachtabsenkung_So.Uhrzeit_Stunde_Ende := 3.5;(*Uhr*)

	Initialisierung.Regelventil_350_Parameter.AutoQuittierung := 0;
	Initialisierung.Regelventil_350_Parameter.Regelung_PI_Kp := 0.265;
	Initialisierung.Regelventil_350_Parameter.Regelung_PI_Tctr := 5000;(*Millisekunden*)
	Initialisierung.Regelventil_350_Parameter.Regelung_PI_Tn := 15000;(*Millisekunden*)
	Initialisierung.Regelventil_350_Parameter.Regelung_Sollw_Max := 70; (*Grad Celsius*)
	Initialisierung.Regelventil_350_Parameter.Regelung_Sollw_Min := 30; (*Grad Celsius*)
	Initialisierung.Regelventil_350_Parameter.Regelung_Sollw_Rampe_Steig_neg := 0.008;(*Einheit: K/s,  0,008 K/s ~ 30 K/h*)
	Initialisierung.Regelventil_350_Parameter.Regelung_Sollw_Rampe_Steig_pos := 0.008;(*Einheit: K/s,  0,008 K/s ~ 30 K/h*)
	Initialisierung.Regelventil_350_Parameter.Stellwert_Stellung_Max := 100;(*Prozent*)
	Initialisierung.Regelventil_350_Parameter.Stellwert_Stellung_Min := 0;(*Prozent*)
	Initialisierung.Regelventil_350_Parameter.Zeit_Nachl := 15000;(*Millisekunden*)
	Initialisierung.Regelventil_350_Parameter.Zeit_Vorl := 15000;(*Millisekunden*)

	Initialisierung.Pumpe_350_Parameter.AutoQuittierung := 0;
	Initialisierung.Pumpe_350_Parameter.Regelung_PI_Kp := 0.265;
	Initialisierung.Pumpe_350_Parameter.Regelung_PI_Tctr := 5000;(*Millisekunden*)
	Initialisierung.Pumpe_350_Parameter.Regelung_PI_Tn := 15000;(*Millisekunden*)
	Initialisierung.Pumpe_350_Parameter.Stellwert_Leistung_Max := 100;(*Prozent*)
	Initialisierung.Pumpe_350_Parameter.Stellwert_Leistung_Min := 50;(*Prozent*)
	Initialisierung.Pumpe_350_Parameter.Zeit_Nachl := 2000;(*Millisekunden*)
	Initialisierung.Pumpe_350_Parameter.Zeit_Vorl := 2000;(*Millisekunden*)


(*Parameter System Thermisches Netz *)
	Initialisierung.System_ThNTZ_Parameter.AutoQuittierung := 0;
	Initialisierung.System_ThNTZ_Parameter.Regelung_PI_Oben_Kp := 1;
	Initialisierung.System_ThNTZ_Parameter.Regelung_PI_Oben_Tctr := 1;(*Millisekunden*)
	Initialisierung.System_ThNTZ_Parameter.Regelung_PI_Oben_Tn := 1;(*Millisekunden*)
	Initialisierung.System_ThNTZ_Parameter.Regelung_Sollw_Max := 95;(*Prozent*)
	Initialisierung.System_ThNTZ_Parameter.Regelung_Sollw_Min := 5;(*Prozent*)
	Initialisierung.System_ThNTZ_Parameter.Stellwert_Leistung_Max := 100;(*Prozent*)
	Initialisierung.System_ThNTZ_Parameter.Stellwert_Leistung_Min := -100;(*Prozent*)
	Initialisierung.System_ThNTZ_Parameter.Temp_Max := 100; (*Grad Celsius*)
	Initialisierung.System_ThNTZ_Parameter.Temp_Min := 0; (*Grad Celsius*)



(*Parameter System Wand- und Deckentemperierung *)

	Initialisierung.System_WDT_Parameter.Temp_Warmwasser_Max := 45 ; (*Grad Celsius*)
	Initialisierung.System_WDT_Parameter.Temp_Warmwasser_Min := 35   ; (*Grad Celsius*)
	Initialisierung.System_WDT_Parameter.Temp_Kaltwasser_Max := 17 ; (*Grad Celsius*)
	Initialisierung.System_WDT_Parameter.Temp_Kaltwasser_Min := 12  ; (*Grad Celsius*)

	(* Heizkurve mit Neigung 0.6 https://www.vaillant.de/heizung/heizung-verstehen/tipps-rund-um-ihre-heizung/vorlauf-rucklauftemperatur/*)
	Initialisierung.System_WDT_Parameter.Kennlinie_Heizung.Temp_Aussen_Max := 15; (*Grad Celsius*)
	Initialisierung.System_WDT_Parameter.Kennlinie_Heizung.Temp_Aussen_Min := -2; (*Grad Celsius*)
	Initialisierung.System_WDT_Parameter.Kennlinie_Heizung.Temp_Vorl_Max := 38; (*Grad Celsius*)
	Initialisierung.System_WDT_Parameter.Kennlinie_Heizung.Temp_Vorl_Min := 25; (*Grad Celsius*)

	Initialisierung.System_WDT_Parameter.Kennlinie_Kuehlung.Temp_Aussen_Max := 40; (*Grad Celsius*)
	Initialisierung.System_WDT_Parameter.Kennlinie_Kuehlung.Temp_Aussen_Min := 25; (*Grad Celsius*)
	Initialisierung.System_WDT_Parameter.Kennlinie_Kuehlung.Temp_Vorl_Max := 22; (*Grad Celsius*)
	Initialisierung.System_WDT_Parameter.Kennlinie_Kuehlung.Temp_Vorl_Min := 20; (*Grad Celsius*)

	Initialisierung.System_WDT_Parameter.AutoQuittierung := 0;
	Initialisierung.System_WDT_Parameter.Temp_Vorl_Max := 41; (*Grad Celsius*)
	Initialisierung.System_WDT_Parameter.Temp_Vorl_Min := 12; (*Grad Celsius*)
	Initialisierung.System_WDT_Parameter.Kennlinie_Tctr := 5000;(*Millisekunden*)
	Initialisierung.System_WDT_Parameter.Systemdruck_Max := 2500;(* mbar *)
	Initialisierung.System_WDT_Parameter.Systemdruck_Min := 500;(* mbar *)

	Initialisierung.System_WDT_Parameter.Nachtabsenkung_Mo.Temp_Absenkung := 10; (*Grad Celsius*)
	Initialisierung.System_WDT_Parameter.Nachtabsenkung_Mo.Uhrzeit_Stunde_Start := 21;(*Uhr*)
	Initialisierung.System_WDT_Parameter.Nachtabsenkung_Mo.Uhrzeit_Stunde_Ende := 3.5;(*Uhr*)
	Initialisierung.System_WDT_Parameter.Nachtabsenkung_Di.Temp_Absenkung := 10; (*Grad Celsius*)
	Initialisierung.System_WDT_Parameter.Nachtabsenkung_Di.Uhrzeit_Stunde_Start := 21;(*Uhr*)
	Initialisierung.System_WDT_Parameter.Nachtabsenkung_Di.Uhrzeit_Stunde_Ende := 3.5;(*Uhr*)
	Initialisierung.System_WDT_Parameter.Nachtabsenkung_Mi.Temp_Absenkung := 10; (*Grad Celsius*)
	Initialisierung.System_WDT_Parameter.Nachtabsenkung_Mi.Uhrzeit_Stunde_Start := 21;(*Uhr*)
	Initialisierung.System_WDT_Parameter.Nachtabsenkung_Mi.Uhrzeit_Stunde_Ende := 3.5;(*Uhr*)
	Initialisierung.System_WDT_Parameter.Nachtabsenkung_Do.Temp_Absenkung := 10; (*Grad Celsius*)
	Initialisierung.System_WDT_Parameter.Nachtabsenkung_Do.Uhrzeit_Stunde_Start := 21;(*Uhr*)
	Initialisierung.System_WDT_Parameter.Nachtabsenkung_Do.Uhrzeit_Stunde_Ende := 3.5;(*Uhr*)
	Initialisierung.System_WDT_Parameter.Nachtabsenkung_Fr.Temp_Absenkung := 10; (*Grad Celsius*)
	Initialisierung.System_WDT_Parameter.Nachtabsenkung_Fr.Uhrzeit_Stunde_Start := 21;(*Uhr*)
	Initialisierung.System_WDT_Parameter.Nachtabsenkung_Fr.Uhrzeit_Stunde_Ende := 3.5;(*Uhr*)
	Initialisierung.System_WDT_Parameter.Nachtabsenkung_Sa.Temp_Absenkung := 10; (*Grad Celsius*)
	Initialisierung.System_WDT_Parameter.Nachtabsenkung_Sa.Uhrzeit_Stunde_Start := 21;(*Uhr*)
	Initialisierung.System_WDT_Parameter.Nachtabsenkung_Sa.Uhrzeit_Stunde_Ende := 3.5;(*Uhr*)
	Initialisierung.System_WDT_Parameter.Nachtabsenkung_So.Temp_Absenkung := 10; (*Grad Celsius*)
	Initialisierung.System_WDT_Parameter.Nachtabsenkung_So.Uhrzeit_Stunde_Start := 21;(*Uhr*)
	Initialisierung.System_WDT_Parameter.Nachtabsenkung_So.Uhrzeit_Stunde_Ende := 3.5;(*Uhr*)

	Initialisierung.Regelventil_500_Parameter.AutoQuittierung := 0;
	Initialisierung.Regelventil_500_Parameter.Regelung_PI_Kp := 0.5;
	Initialisierung.Regelventil_500_Parameter.Regelung_PI_Tctr := 5000;(*Millisekunden*)
	Initialisierung.Regelventil_500_Parameter.Regelung_PI_Tn := 15000;(*Millisekunden*)
	Initialisierung.Regelventil_500_Parameter.Regelung_Sollw_Max := 45; (*Grad Celsius*)
	Initialisierung.Regelventil_500_Parameter.Regelung_Sollw_Min := 15; (*Grad Celsius*)
	Initialisierung.Regelventil_500_Parameter.Regelung_Sollw_Rampe_Steig_neg := 0.0005;(*Einheit: K/s,  0,0005 K/s ~ 2 K/h*)
	Initialisierung.Regelventil_500_Parameter.Regelung_Sollw_Rampe_Steig_pos := 0.0005;(*Einheit: K/s,  0,0005 K/s ~ 2 K/h*)
	Initialisierung.Regelventil_500_Parameter.Stellwert_Stellung_Max := 100;(*Prozent*)
	Initialisierung.Regelventil_500_Parameter.Stellwert_Stellung_Min := 0;(*Prozent*)
	Initialisierung.Regelventil_500_Parameter.Zeit_Nachl := 15000;(*Millisekunden*)
	Initialisierung.Regelventil_500_Parameter.Zeit_Vorl := 15000;(*Millisekunden*)

	Initialisierung.Regelventil_541_Parameter.AutoQuittierung := 0;
	Initialisierung.Regelventil_541_Parameter.Regelung_PI_Kp := 0.265;
	Initialisierung.Regelventil_541_Parameter.Regelung_PI_Tctr := 5000;(*Millisekunden*)
	Initialisierung.Regelventil_541_Parameter.Regelung_PI_Tn := 15000;(*Millisekunden*)
	Initialisierung.Regelventil_541_Parameter.Regelung_Sollw_Max := 35; (*Grad Celsius*)
	Initialisierung.Regelventil_541_Parameter.Regelung_Sollw_Min := 15; (*Grad Celsius*)
	Initialisierung.Regelventil_541_Parameter.Regelung_Sollw_Rampe_Steig_neg := 0.0005;(*Einheit: K/s,  0,0005 K/s ~ 2 K/h*)
	Initialisierung.Regelventil_541_Parameter.Regelung_Sollw_Rampe_Steig_pos := 0.0005;(*Einheit: K/s,  0,0005 K/s ~ 2 K/h*)
	Initialisierung.Regelventil_541_Parameter.Stellwert_Stellung_Max := 100;(*Prozent*)
	Initialisierung.Regelventil_541_Parameter.Stellwert_Stellung_Min := 0;(*Prozent*)
	Initialisierung.Regelventil_541_Parameter.Zeit_Nachl := 15000;(*Millisekunden*)
	Initialisierung.Regelventil_541_Parameter.Zeit_Vorl := 15000;(*Millisekunden*)

	Initialisierung.Regelventil_542_Parameter.AutoQuittierung := 0;
	Initialisierung.Regelventil_542_Parameter.Regelung_PI_Kp := 0.265;
	Initialisierung.Regelventil_542_Parameter.Regelung_PI_Tctr := 5000;(*Millisekunden*)
	Initialisierung.Regelventil_542_Parameter.Regelung_PI_Tn := 15000;(*Millisekunden*)
	Initialisierung.Regelventil_542_Parameter.Regelung_Sollw_Max := 35; (*Grad Celsius*)
	Initialisierung.Regelventil_542_Parameter.Regelung_Sollw_Min := 15; (*Grad Celsius*)
	Initialisierung.Regelventil_542_Parameter.Regelung_Sollw_Rampe_Steig_neg := 0.0005;(*Einheit: K/s,  0,0005 K/s ~ 2 K/h*)
	Initialisierung.Regelventil_542_Parameter.Regelung_Sollw_Rampe_Steig_pos := 0.0005;(*Einheit: K/s,  0,0005 K/s ~ 2 K/h*)
	Initialisierung.Regelventil_542_Parameter.Stellwert_Stellung_Max := 100;(*Prozent*)
	Initialisierung.Regelventil_542_Parameter.Stellwert_Stellung_Min := 0;(*Prozent*)
	Initialisierung.Regelventil_542_Parameter.Zeit_Nachl := 15000;(*Millisekunden*)
	Initialisierung.Regelventil_542_Parameter.Zeit_Vorl := 15000;(*Millisekunden*)

	Initialisierung.Regelventil_543_Parameter.AutoQuittierung := 0;
	Initialisierung.Regelventil_543_Parameter.Regelung_PI_Kp := 0.265;
	Initialisierung.Regelventil_543_Parameter.Regelung_PI_Tctr := 5000;(*Millisekunden*)
	Initialisierung.Regelventil_543_Parameter.Regelung_PI_Tn := 15000;(*Millisekunden*)
	Initialisierung.Regelventil_543_Parameter.Regelung_Sollw_Max := 35; (*Grad Celsius*)
	Initialisierung.Regelventil_543_Parameter.Regelung_Sollw_Min := 15; (*Grad Celsius*)
	Initialisierung.Regelventil_543_Parameter.Regelung_Sollw_Rampe_Steig_neg := 0.0005;(*Einheit: K/s,  0,0005 K/s ~ 2 K/h*)
	Initialisierung.Regelventil_543_Parameter.Regelung_Sollw_Rampe_Steig_pos := 0.0005;(*Einheit: K/s,  0,0005 K/s ~ 2 K/h*)
	Initialisierung.Regelventil_543_Parameter.Stellwert_Stellung_Max := 100;(*Prozent*)
	Initialisierung.Regelventil_543_Parameter.Stellwert_Stellung_Min := 0;(*Prozent*)
	Initialisierung.Regelventil_543_Parameter.Zeit_Nachl := 15000;(*Millisekunden*)
	Initialisierung.Regelventil_543_Parameter.Zeit_Vorl := 15000;(*Millisekunden*)


	Initialisierung.Regelventil_551_Parameter.AutoQuittierung := 0;
	Initialisierung.Regelventil_551_Parameter.Regelung_PI_Kp := 0.265;
	Initialisierung.Regelventil_551_Parameter.Regelung_PI_Tctr := 5000;(*Millisekunden*)
	Initialisierung.Regelventil_551_Parameter.Regelung_PI_Tn := 15000;(*Millisekunden*)
	Initialisierung.Regelventil_551_Parameter.Regelung_Sollw_Max := 35; (*Grad Celsius*)
	Initialisierung.Regelventil_551_Parameter.Regelung_Sollw_Min := 15; (*Grad Celsius*)
	Initialisierung.Regelventil_551_Parameter.Regelung_Sollw_Rampe_Steig_neg := 0.0005;(*Einheit: K/s,  0,0005 K/s ~ 2 K/h*)
	Initialisierung.Regelventil_551_Parameter.Regelung_Sollw_Rampe_Steig_pos := 0.0005;(*Einheit: K/s,  0,0005 K/s ~ 2 K/h*)
	Initialisierung.Regelventil_551_Parameter.Stellwert_Stellung_Max := 100;(*Prozent*)
	Initialisierung.Regelventil_551_Parameter.Stellwert_Stellung_Min := 0;(*Prozent*)
	Initialisierung.Regelventil_551_Parameter.Zeit_Nachl := 15000;(*Millisekunden*)
	Initialisierung.Regelventil_551_Parameter.Zeit_Vorl := 15000;(*Millisekunden*)

	Initialisierung.Regelventil_552_Parameter.AutoQuittierung := 0;
	Initialisierung.Regelventil_552_Parameter.Regelung_PI_Kp := 0.265;
	Initialisierung.Regelventil_552_Parameter.Regelung_PI_Tctr := 5000;(*Millisekunden*)
	Initialisierung.Regelventil_552_Parameter.Regelung_PI_Tn := 15000;(*Millisekunden*)
	Initialisierung.Regelventil_552_Parameter.Regelung_Sollw_Max := 35; (*Grad Celsius*)
	Initialisierung.Regelventil_552_Parameter.Regelung_Sollw_Min := 15; (*Grad Celsius*)
	Initialisierung.Regelventil_552_Parameter.Regelung_Sollw_Rampe_Steig_neg := 0.0005;(*Einheit: K/s,  0,0005 K/s ~ 2 K/h*)
	Initialisierung.Regelventil_552_Parameter.Regelung_Sollw_Rampe_Steig_pos := 0.0005;(*Einheit: K/s,  0,0005 K/s ~ 2 K/h*)
	Initialisierung.Regelventil_552_Parameter.Stellwert_Stellung_Max := 100;(*Prozent*)
	Initialisierung.Regelventil_552_Parameter.Stellwert_Stellung_Min := 0;(*Prozent*)
	Initialisierung.Regelventil_552_Parameter.Zeit_Nachl := 15000;(*Millisekunden*)
	Initialisierung.Regelventil_552_Parameter.Zeit_Vorl := 15000;(*Millisekunden*)

	Initialisierung.Regelventil_553_Parameter.AutoQuittierung := 0;
	Initialisierung.Regelventil_553_Parameter.Regelung_PI_Kp := 0.265;
	Initialisierung.Regelventil_553_Parameter.Regelung_PI_Tctr := 5000;(*Millisekunden*)
	Initialisierung.Regelventil_553_Parameter.Regelung_PI_Tn := 15000;(*Millisekunden*)
	Initialisierung.Regelventil_553_Parameter.Regelung_Sollw_Max := 35; (*Grad Celsius*)
	Initialisierung.Regelventil_553_Parameter.Regelung_Sollw_Min := 15; (*Grad Celsius*)
	Initialisierung.Regelventil_553_Parameter.Regelung_Sollw_Rampe_Steig_neg := 0.0005;(*Einheit: K/s,  0,0005 K/s ~ 2 K/h*)
	Initialisierung.Regelventil_553_Parameter.Regelung_Sollw_Rampe_Steig_pos := 0.0005;(*Einheit: K/s,  0,0005 K/s ~ 2 K/h*)
	Initialisierung.Regelventil_553_Parameter.Stellwert_Stellung_Max := 100;(*Prozent*)
	Initialisierung.Regelventil_553_Parameter.Stellwert_Stellung_Min := 0;(*Prozent*)
	Initialisierung.Regelventil_553_Parameter.Zeit_Nachl := 15000;(*Millisekunden*)
	Initialisierung.Regelventil_553_Parameter.Zeit_Vorl := 15000;(*Millisekunden*)


	Initialisierung.Regelventil_561_Parameter.AutoQuittierung := 0;
	Initialisierung.Regelventil_561_Parameter.Regelung_PI_Kp := 0.265;
	Initialisierung.Regelventil_561_Parameter.Regelung_PI_Tctr := 5000;(*Millisekunden*)
	Initialisierung.Regelventil_561_Parameter.Regelung_PI_Tn := 15000;(*Millisekunden*)
	Initialisierung.Regelventil_561_Parameter.Regelung_Sollw_Max := 35; (*Grad Celsius*)
	Initialisierung.Regelventil_561_Parameter.Regelung_Sollw_Min := 15; (*Grad Celsius*)
	Initialisierung.Regelventil_561_Parameter.Regelung_Sollw_Rampe_Steig_neg := 0.0005;(*Einheit: K/s,  0,0005 K/s ~ 2 K/h*)
	Initialisierung.Regelventil_561_Parameter.Regelung_Sollw_Rampe_Steig_pos := 0.0005;(*Einheit: K/s,  0,0005 K/s ~ 2 K/h*)
	Initialisierung.Regelventil_561_Parameter.Stellwert_Stellung_Max := 100;(*Prozent*)
	Initialisierung.Regelventil_561_Parameter.Stellwert_Stellung_Min := 0;(*Prozent*)
	Initialisierung.Regelventil_561_Parameter.Zeit_Nachl := 15000;(*Millisekunden*)
	Initialisierung.Regelventil_561_Parameter.Zeit_Vorl := 15000;(*Millisekunden*)

	Initialisierung.Regelventil_562_Parameter.AutoQuittierung := 0;
	Initialisierung.Regelventil_562_Parameter.Regelung_PI_Kp := 0.265;
	Initialisierung.Regelventil_562_Parameter.Regelung_PI_Tctr := 5000;(*Millisekunden*)
	Initialisierung.Regelventil_562_Parameter.Regelung_PI_Tn := 15000;(*Millisekunden*)
	Initialisierung.Regelventil_562_Parameter.Regelung_Sollw_Max := 35; (*Grad Celsius*)
	Initialisierung.Regelventil_562_Parameter.Regelung_Sollw_Min := 15; (*Grad Celsius*)
	Initialisierung.Regelventil_562_Parameter.Regelung_Sollw_Rampe_Steig_neg := 0.0005;(*Einheit: K/s,  0,0005 K/s ~ 2 K/h*)
	Initialisierung.Regelventil_562_Parameter.Regelung_Sollw_Rampe_Steig_pos := 0.0005;(*Einheit: K/s,  0,0005 K/s ~ 2 K/h*)
	Initialisierung.Regelventil_562_Parameter.Stellwert_Stellung_Max := 100;(*Prozent*)
	Initialisierung.Regelventil_562_Parameter.Stellwert_Stellung_Min := 0;(*Prozent*)
	Initialisierung.Regelventil_562_Parameter.Zeit_Nachl := 15000;(*Millisekunden*)
	Initialisierung.Regelventil_562_Parameter.Zeit_Vorl := 15000;(*Millisekunden*)

	Initialisierung.Regelventil_563_Parameter.AutoQuittierung := 0;
	Initialisierung.Regelventil_563_Parameter.Regelung_PI_Kp := 0.265;
	Initialisierung.Regelventil_563_Parameter.Regelung_PI_Tctr := 5000;(*Millisekunden*)
	Initialisierung.Regelventil_563_Parameter.Regelung_PI_Tn := 15000;(*Millisekunden*)
	Initialisierung.Regelventil_563_Parameter.Regelung_Sollw_Max := 35; (*Grad Celsius*)
	Initialisierung.Regelventil_563_Parameter.Regelung_Sollw_Min := 15; (*Grad Celsius*)
	Initialisierung.Regelventil_563_Parameter.Regelung_Sollw_Rampe_Steig_neg := 0.0005;(*Einheit: K/s,  0,0005 K/s ~ 2 K/h*)
	Initialisierung.Regelventil_563_Parameter.Regelung_Sollw_Rampe_Steig_pos := 0.0005;(*Einheit: K/s,  0,0005 K/s ~ 2 K/h*)
	Initialisierung.Regelventil_563_Parameter.Stellwert_Stellung_Max := 100;(*Prozent*)
	Initialisierung.Regelventil_563_Parameter.Stellwert_Stellung_Min := 0;(*Prozent*)
	Initialisierung.Regelventil_563_Parameter.Zeit_Nachl := 15000;(*Millisekunden*)
	Initialisierung.Regelventil_563_Parameter.Zeit_Vorl := 15000;(*Millisekunden*)

	Initialisierung.Regelventil_571_Parameter.AutoQuittierung := 0;
	Initialisierung.Regelventil_571_Parameter.Regelung_PI_Kp := 0.265;
	Initialisierung.Regelventil_571_Parameter.Regelung_PI_Tctr := 5000;(*Millisekunden*)
	Initialisierung.Regelventil_571_Parameter.Regelung_PI_Tn := 15000;(*Millisekunden*)
	Initialisierung.Regelventil_571_Parameter.Regelung_Sollw_Max := 35; (*Grad Celsius*)
	Initialisierung.Regelventil_571_Parameter.Regelung_Sollw_Min := 15; (*Grad Celsius*)
	Initialisierung.Regelventil_571_Parameter.Regelung_Sollw_Rampe_Steig_neg := 0.0005;(*Einheit: K/s,  0,0005 K/s ~ 2 K/h*)
	Initialisierung.Regelventil_571_Parameter.Regelung_Sollw_Rampe_Steig_pos := 0.0005;(*Einheit: K/s,  0,0005 K/s ~ 2 K/h*)
	Initialisierung.Regelventil_571_Parameter.Stellwert_Stellung_Max := 100;(*Prozent*)
	Initialisierung.Regelventil_571_Parameter.Stellwert_Stellung_Min := 0;(*Prozent*)
	Initialisierung.Regelventil_571_Parameter.Zeit_Nachl := 15000;(*Millisekunden*)
	Initialisierung.Regelventil_571_Parameter.Zeit_Vorl := 15000;(*Millisekunden*)

	Initialisierung.Regelventil_572_Parameter.AutoQuittierung := 0;
	Initialisierung.Regelventil_572_Parameter.Regelung_PI_Kp := 0.265;
	Initialisierung.Regelventil_572_Parameter.Regelung_PI_Tctr := 5000;(*Millisekunden*)
	Initialisierung.Regelventil_572_Parameter.Regelung_PI_Tn := 15000;(*Millisekunden*)
	Initialisierung.Regelventil_572_Parameter.Regelung_Sollw_Max := 35; (*Grad Celsius*)
	Initialisierung.Regelventil_572_Parameter.Regelung_Sollw_Min := 15; (*Grad Celsius*)
	Initialisierung.Regelventil_572_Parameter.Regelung_Sollw_Rampe_Steig_neg := 0.0005;(*Einheit: K/s,  0,0005 K/s ~ 2 K/h*)
	Initialisierung.Regelventil_572_Parameter.Regelung_Sollw_Rampe_Steig_pos := 0.0005;(*Einheit: K/s,  0,0005 K/s ~ 2 K/h*)
	Initialisierung.Regelventil_572_Parameter.Stellwert_Stellung_Max := 100;(*Prozent*)
	Initialisierung.Regelventil_572_Parameter.Stellwert_Stellung_Min := 0;(*Prozent*)
	Initialisierung.Regelventil_572_Parameter.Zeit_Nachl := 15000;(*Millisekunden*)
	Initialisierung.Regelventil_572_Parameter.Zeit_Vorl := 15000;(*Millisekunden*)

	Initialisierung.Regelventil_573_Parameter.AutoQuittierung := 0;
	Initialisierung.Regelventil_573_Parameter.Regelung_PI_Kp := 0.265;
	Initialisierung.Regelventil_573_Parameter.Regelung_PI_Tctr := 5000;(*Millisekunden*)
	Initialisierung.Regelventil_573_Parameter.Regelung_PI_Tn := 15000;(*Millisekunden*)
	Initialisierung.Regelventil_573_Parameter.Regelung_Sollw_Max := 35; (*Grad Celsius*)
	Initialisierung.Regelventil_573_Parameter.Regelung_Sollw_Min := 15; (*Grad Celsius*)
	Initialisierung.Regelventil_573_Parameter.Regelung_Sollw_Rampe_Steig_neg := 0.0005;(*Einheit: K/s,  0,0005 K/s ~ 2 K/h*)
	Initialisierung.Regelventil_573_Parameter.Regelung_Sollw_Rampe_Steig_pos := 0.0005;(*Einheit: K/s,  0,0005 K/s ~ 2 K/h*)
	Initialisierung.Regelventil_573_Parameter.Stellwert_Stellung_Max := 100;(*Prozent*)
	Initialisierung.Regelventil_573_Parameter.Stellwert_Stellung_Min := 0;(*Prozent*)
	Initialisierung.Regelventil_573_Parameter.Zeit_Nachl := 15000;(*Millisekunden*)
	Initialisierung.Regelventil_573_Parameter.Zeit_Vorl := 15000;(*Millisekunden*)

	Initialisierung.Stellventil_401_402_Parameter.AutoQuittierung := 0;
	Initialisierung.Stellventil_401_402_Parameter.Zeit_Stellen0 := 10000;(*Millisekunden*)
	Initialisierung.Stellventil_401_402_Parameter.Zeit_Stellen1 := 10000;(*Millisekunden*)

	Initialisierung.Stellventil_403_404_Parameter.AutoQuittierung := 0;
	Initialisierung.Stellventil_403_404_Parameter.Zeit_Stellen0 := 10000;(*Millisekunden*)
	Initialisierung.Stellventil_403_404_Parameter.Zeit_Stellen1 := 10000;(*Millisekunden*)

	Initialisierung.Stellventil_504_505_Parameter.AutoQuittierung := 0;
	Initialisierung.Stellventil_504_505_Parameter.Zeit_Stellen0 := 10000;(*Millisekunden*)
	Initialisierung.Stellventil_504_505_Parameter.Zeit_Stellen1 := 10000;(*Millisekunden*)

	Initialisierung.Pumpe_405_Parameter.AutoQuittierung := 0;
	Initialisierung.Pumpe_405_Parameter.Regelung_PI_Kp := 0.265;
	Initialisierung.Pumpe_405_Parameter.Regelung_PI_Tctr := 5000;(*Millisekunden*)
	Initialisierung.Pumpe_405_Parameter.Regelung_PI_Tn := 15000;(*Millisekunden*)
	Initialisierung.Pumpe_405_Parameter.Stellwert_Leistung_Max := 100;(*Prozent*)
	Initialisierung.Pumpe_405_Parameter.Stellwert_Leistung_Min := 50;(*Prozent*)
	Initialisierung.Pumpe_405_Parameter.Zeit_Nachl := 2000;(*Millisekunden*)
	Initialisierung.Pumpe_405_Parameter.Zeit_Vorl := 2000;(*Millisekunden*)

	Initialisierung.Pumpe_500_Parameter.AutoQuittierung := 0;
	Initialisierung.Pumpe_500_Parameter.Regelung_PI_Kp := 0.265;
	Initialisierung.Pumpe_500_Parameter.Regelung_PI_Tctr := 5000;(*Millisekunden*)
	Initialisierung.Pumpe_500_Parameter.Regelung_PI_Tn := 15000;(*Millisekunden*)
	Initialisierung.Pumpe_500_Parameter.Stellwert_Leistung_Max := 100;(*Prozent*)
	Initialisierung.Pumpe_500_Parameter.Stellwert_Leistung_Min := 50;(*Prozent*)
	Initialisierung.Pumpe_500_Parameter.Zeit_Nachl := 2000;(*Millisekunden*)
	Initialisierung.Pumpe_500_Parameter.Zeit_Vorl := 2000;(*Millisekunden*)

(*Parameter System Wärmetauscher *)
	Initialisierung.System_WT_HWW_Parameter.AutoQuittierung := 0;

	Initialisierung.Stellventil_215_Parameter.AutoQuittierung := 0;
	Initialisierung.Stellventil_215_Parameter.Zeit_Stellen0 := 75000;(*Millisekunden*)
	Initialisierung.Stellventil_215_Parameter.Zeit_Stellen1 := 20000;(*Millisekunden*)

	Initialisierung.Stellventil_315_Parameter.AutoQuittierung := 0;
	Initialisierung.Stellventil_315_Parameter.Zeit_Stellen0 := 75000;(*Millisekunden*)
	Initialisierung.Stellventil_315_Parameter.Zeit_Stellen1 := 20000;(*Millisekunden*)

	Initialisierung.Pumpe_215_Parameter.AutoQuittierung := 0;
	Initialisierung.Pumpe_215_Parameter.Regelung_PI_Kp := 0.265;
	Initialisierung.Pumpe_215_Parameter.Regelung_PI_Tctr := 5000;(*Millisekunden*)
	Initialisierung.Pumpe_215_Parameter.Regelung_PI_Tn := 15000;(*Millisekunden*)
	Initialisierung.Pumpe_215_Parameter.Stellwert_Leistung_Max := 100;(*Prozent*)
	Initialisierung.Pumpe_215_Parameter.Stellwert_Leistung_Min := 50;(*Prozent*)
	Initialisierung.Pumpe_215_Parameter.Zeit_Nachl := 2000;(*Millisekunden*)
	Initialisierung.Pumpe_215_Parameter.Zeit_Vorl := 2000;(*Millisekunden*)

	Initialisierung.Pumpe_315_Parameter.AutoQuittierung := 0;
	Initialisierung.Pumpe_315_Parameter.Regelung_PI_Kp := 0.265;
	Initialisierung.Pumpe_315_Parameter.Regelung_PI_Tctr := 5000;(*Millisekunden*)
	Initialisierung.Pumpe_315_Parameter.Regelung_PI_Tn := 15000;(*Millisekunden*)
	Initialisierung.Pumpe_315_Parameter.Stellwert_Leistung_Max := 100;(*Prozent*)
	Initialisierung.Pumpe_315_Parameter.Stellwert_Leistung_Min := 50;(*Prozent*)
	Initialisierung.Pumpe_315_Parameter.Zeit_Nachl := 2000;(*Millisekunden*)
	Initialisierung.Pumpe_315_Parameter.Zeit_Vorl := 2000;(*Millisekunden*)

	Initialisierung.Regelventil_215_Parameter.AutoQuittierung := 0;
	Initialisierung.Regelventil_215_Parameter.Regelung_PI_Kp := 0.265;
	Initialisierung.Regelventil_215_Parameter.Regelung_PI_Tctr := 5000;(*Millisekunden*)
	Initialisierung.Regelventil_215_Parameter.Regelung_PI_Tn := 15000;(*Millisekunden*)
	Initialisierung.Regelventil_215_Parameter.Regelung_Sollw_Max := 35; (*Grad Celsius*)
	Initialisierung.Regelventil_215_Parameter.Regelung_Sollw_Min := 15; (*Grad Celsius*)
	Initialisierung.Regelventil_215_Parameter.Regelung_Sollw_Rampe_Steig_neg := 0.0005;(*Einheit: K/s,  0,0005 K/s ~ 2 K/h*)
	Initialisierung.Regelventil_215_Parameter.Regelung_Sollw_Rampe_Steig_pos := 0.0005;(*Einheit: K/s,  0,0005 K/s ~ 2 K/h*)
	Initialisierung.Regelventil_215_Parameter.Stellwert_Stellung_Max := 100;(*Prozent*)
	Initialisierung.Regelventil_215_Parameter.Stellwert_Stellung_Min := 0;(*Prozent*)
	Initialisierung.Regelventil_215_Parameter.Zeit_Nachl := 15000;(*Millisekunden*)
	Initialisierung.Regelventil_215_Parameter.Zeit_Vorl := 15000;(*Millisekunden*)

(*Parameter System Wärmepumpe *)
	Initialisierung.System_WP_946_Parameter.AutoQuittierung := 0;

	Initialisierung.Stellventil_146_Parameter.AutoQuittierung := 0;
	Initialisierung.Stellventil_146_Parameter.Zeit_Stellen0 := 10000;(*Millisekunden*)
	Initialisierung.Stellventil_146_Parameter.Zeit_Stellen1 := 10000;(*Millisekunden*)

	Initialisierung.Stellventil_246_Parameter.AutoQuittierung := 0;
	Initialisierung.Stellventil_246_Parameter.Zeit_Stellen0 := 10000;(*Millisekunden*)
	Initialisierung.Stellventil_246_Parameter.Zeit_Stellen1 := 10000;(*Millisekunden*)

	Initialisierung.Anlage_WP_946_Parameter.AutoQuittierung := 0;
	Initialisierung.Anlage_WP_946_Parameter.Temp_Kaltwasser 	:= 17; (*Grad Celsius*)
	Initialisierung.Anlage_WP_946_Parameter.Temp_Kaltwasser_Max := 20; (*Grad Celsius*)
	Initialisierung.Anlage_WP_946_Parameter.Temp_Kaltwasser_Min := 8; (*Grad Celsius*)

	Initialisierung.Anlage_WP_946_Parameter.Zeit_Nachl := 900000; (*Millisekunden*)(*15 min*)
	Initialisierung.Anlage_WP_946_Parameter.Zeit_Vorl := 60000;(*Millisekunden*)

END_FUNCTION_BLOCK

// ---- POUs/Checks/CheckBounds.TcPOU
FUNCTION CheckBounds : DINT
VAR_INPUT
	index, lower, upper 	: DINT;
END_VAR
VAR
END_VAR

IF index<lower THEN
	CheckBounds_ErrCnt := CheckBounds_ErrCnt + 1;
	CheckBounds := lower;
ELSIF index>upper THEN
	CheckBounds_ErrCnt := CheckBounds_ErrCnt + 1;
	CheckBounds := upper;
ELSE
	CheckBounds := index;
END_IF

END_FUNCTION

// ---- POUs/Checks/CheckDivDWord.TcPOU
FUNCTION CheckDivDWord : DWORD
VAR_INPUT
	divisor				: DWORD;
END_VAR
VAR
END_VAR

IF divisor = 0 THEN
	CheckDWordZeroDiv_ErrCnt := CheckDWordZeroDiv_ErrCnt + 1;
	CheckDivDWord := 1;
ELSE
	CheckDivDWord := divisor;
END_IF

END_FUNCTION

// ---- POUs/Checks/CheckDivReal.TcPOU
FUNCTION CheckDivReal : REAL
VAR_INPUT
	divisor		 		: REAL;
END_VAR
VAR
END_VAR

IF divisor = 0 THEN
	CheckRealZeroDiv_ErrCnt := CheckRealZeroDiv_ErrCnt + 1;
	CheckDivReal := 1;
ELSE
	CheckDivReal := divisor;
END_IF

END_FUNCTION

// ---- POUs/Checks/CheckDivWord.TcPOU
FUNCTION CheckDivWord : WORD
VAR_INPUT
	divisor				: WORD;
END_VAR
VAR
END_VAR

IF divisor = 0 THEN
	CheckWordZeroDiv_ErrCnt:= CheckWordZeroDiv_ErrCnt + 1;
	CheckDivWord := 1;
ELSE
	CheckDivWord := divisor;
END_IF

END_FUNCTION

// ---- POUs/Checks/CheckRangeUnsigned.TcPOU
FUNCTION CheckRangeUnsigned : UDINT
VAR_INPUT
    value, lower, upper: UDINT;
END_VAR
VAR
END_VAR

IF (value < lower) THEN
	CheckRangeUnSigned_ErrCnt := CheckRangeUnsigned_ErrCnt + 1;
	CheckRangeUnsigned := lower;
ELSIF(value > upper) THEN
	CheckRangeUnsigned_ErrCnt := CheckRangeUnsigned_ErrCnt + 1;
	CheckRangeUnsigned := upper;
ELSE
	CheckRangeUnsigned := value;
END_IF

END_FUNCTION

// ---- POUs/Einzelanlagen/Ampel/FB_Ampel_Out.TcPOU
FUNCTION_BLOCK FB_Ampel_Out
VAR_INPUT
	Stellung_Rot		: BOOL;
	Stellung_Orange		: BOOL;
	Stellung_Gruen		: BOOL;
	Stellung_Blau		: BOOL;
	Stellung_Buzz		: BOOL;
	Zustand				: ST_Ampel_Zustand;
END_VAR
VAR_OUTPUT
	OUT_Stellung_Rot			: BOOL;
	OUT_Stellung_Orange			: BOOL;
	OUT_Stellung_Gruen			: BOOL;
	OUT_Stellung_Blau			: BOOL;
	OUT_Stellung_Buzz			: BOOL;
END_VAR
VAR
END_VAR

OUT_Stellung_Rot			:= Stellung_Rot;
OUT_Stellung_Orange			:= Stellung_Orange;
OUT_Stellung_Gruen			:= Stellung_Gruen;
OUT_Stellung_Blau			:= Stellung_Blau;
OUT_Stellung_Buzz			:= Stellung_Buzz;

END_FUNCTION_BLOCK

// ---- POUs/Einzelanlagen/Drucksensor/FB_DS.TcPOU
FUNCTION_BLOCK FB_DS
VAR_INPUT
END_VAR
VAR_OUTPUT
	{attribute 'OPC.UA.DA' := '1'}Parameter		: ST_DS_Parameter;	
	{attribute 'OPC.UA.DA' := '1'}Zustand			: ST_DS_Zustand; 
END_VAR
VAR
	Zustandscheck	: FB_DS_Zustandscheck;

	LeseDaten		: FB_DS_Input;

	IN_Status		AT %I*: USINT;
	IN_Druck		AT%I* : INT;

END_VAR

LeseDaten(IN_Status := IN_Status, IN_Druck := IN_Druck); // FB_DS_Input
Zustand.Druck := LeseDaten.Druck;
Zustandscheck(Parameter := Parameter, Zustand := Zustand); // FB_DS_Zustandscheck

END_FUNCTION_BLOCK

// ---- POUs/Einzelanlagen/Drucksensor/FB_DS_Zustandscheck.TcPOU
FUNCTION_BLOCK FB_DS_Zustandscheck
VAR_IN_OUT
	Zustand			: ST_DS_Zustand;
END_VAR
VAR_INPUT
	Parameter		:ST_DS_Parameter;
END_VAR
VAR_OUTPUT
END_VAR
VAR
END_VAR

(*
	Warnung_Code
		0:	Allgemein Warnung Pufferspeicher
		2:	Grenztemperaturen unter- oder ueberschritten
*)

(* Interne Stoerungen / Warnungen *)
(* Warnung - Grenztemperaturen unter- oder ueberschritten *)
Zustand.Warnung_Code.2	:= Zustand.Druck > Parameter.Druck_Max OR Zustand.Druck < Parameter.Druck_Min;

(* Warnmeldung *)
IF Zustand.Warnung_Code > 0 THEN
	Zustand.Warnung := TRUE;
ELSE
	Zustand.Warnung := FALSE;
END_IF;

END_FUNCTION_BLOCK

// ---- POUs/Einzelanlagen/Drucksensor/FB_DS_Input.TcPOU
FUNCTION_BLOCK FB_DS_Input
VAR_INPUT
	IN_Status		:USINT;
	IN_Druck		:INT;
END_VAR
VAR_OUTPUT
	Status			: USINT;
	Druck			: REAL;
END_VAR
VAR
	(*IN_Druck_Buffer : FB_BUFFER_INT_TO_REAL;*)

	VAR_Druck : REAL;
END_VAR

Status 		:= IN_Status;

(*IN_Druck_Buffer(raw_input := IN_Druck);
Druck	:= IN_Druck_Buffer.real_output;*)

VAR_Druck	 := IN_Druck;
Druck := VAR_Druck * 0.1831 ;  (* skaliert [0,32767] auf [0,6000] *)

END_FUNCTION_BLOCK

// ---- POUs/Einzelanlagen/Fenster/FB_Fenster_Logik.TcPOU
FUNCTION_BLOCK FB_Fenster_Logik
VAR_IN_OUT
	Steuerung	: ST_Fenster_Steuerung;
	Zustand		: ST_Fenster_Zustand;
END_VAR
VAR_INPUT
	Parameter	: ST_Fenster_Parameter;
END_VAR
VAR_OUTPUT
END_VAR
VAR
END_VAR

